{region " SIGNAL AREA : NAME->C_Pnt_Hv_Off LENGTH->2 STARTBIT :22"}
_FB_CanTx_Message_Unpack_450.S_Bit_22		:= (GVL.IOVD.C_Pnt_Hv_Off.x OR GVL.IOVD.C_Pnt_Hv_Off.na) AND NOT GVL.IOVD.C_Pnt_Hv_Off.e; 
_FB_CanTx_Message_Unpack_450.S_Bit_23		:= NOT GVL.IOVD.C_Pnt_Hv_Off.v OR GVL.IOVD.C_Pnt_Hv_Off.na OR GVL.IOVD.C_Pnt_Hv_Off.e; 
{endregion}

{region " SIGNAL AREA : NAME->C_Bat_Lo_Hv_Off LENGTH->2 STARTBIT :24"}
_FB_CanTx_Message_Unpack_450.S_Bit_24		:= (GVL.IOVD.C_Bat_Lo_Hv_Off.x OR GVL.IOVD.C_Bat_Lo_Hv_Off.na) AND NOT GVL.IOVD.C_Bat_Lo_Hv_Off.e; 
_FB_CanTx_Message_Unpack_450.S_Bit_25		:= NOT GVL.IOVD.C_Bat_Lo_Hv_Off.v OR GVL.IOVD.C_Bat_Lo_Hv_Off.na OR GVL.IOVD.C_Bat_Lo_Hv_Off.e; 
{endregion}

{region " SIGNAL AREA : NAME->C_Tm_Hv_Off LENGTH->2 STARTBIT :26"}
_FB_CanTx_Message_Unpack_450.S_Bit_26		:= (GVL.IOVD.C_Tm_Hv_Off.x OR GVL.IOVD.C_Tm_Hv_Off.na) AND NOT GVL.IOVD.C_Tm_Hv_Off.e; 
_FB_CanTx_Message_Unpack_450.S_Bit_27		:= NOT GVL.IOVD.C_Tm_Hv_Off.v OR GVL.IOVD.C_Tm_Hv_Off.na OR GVL.IOVD.C_Tm_Hv_Off.e; 
{endregion}

{region " SIGNAL AREA : NAME->C_Diag_Hv_Off LENGTH->2 STARTBIT :28"}
_FB_CanTx_Message_Unpack_450.S_Bit_28		:= (GVL.IOVD.C_Diag_Hv_Off.x OR GVL.IOVD.C_Diag_Hv_Off.na) AND NOT GVL.IOVD.C_Diag_Hv_Off.e; 
_FB_CanTx_Message_Unpack_450.S_Bit_29		:= NOT GVL.IOVD.C_Diag_Hv_Off.v OR GVL.IOVD.C_Diag_Hv_Off.na OR GVL.IOVD.C_Diag_Hv_Off.e; 
{endregion}

{region " SIGNAL AREA : NAME->C_Hv_On LENGTH->2 STARTBIT :32"}
_FB_CanTx_Message_Unpack_450.S_Bit_32		:= (GVL.IOVD.C_Hv_On.x OR GVL.IOVD.C_Hv_On.na) AND NOT GVL.IOVD.C_Hv_On.e; 
_FB_CanTx_Message_Unpack_450.S_Bit_33		:= NOT GVL.IOVD.C_Hv_On.v OR GVL.IOVD.C_Hv_On.na OR GVL.IOVD.C_Hv_On.e; 
{endregion}

{region " SIGNAL AREA : NAME->C_Hv_Off LENGTH->2 STARTBIT :34"}
_FB_CanTx_Message_Unpack_450.S_Bit_34		:= (GVL.IOVD.C_Hv_Off.x OR GVL.IOVD.C_Hv_Off.na) AND NOT GVL.IOVD.C_Hv_Off.e; 
_FB_CanTx_Message_Unpack_450.S_Bit_35		:= NOT GVL.IOVD.C_Hv_Off.v OR GVL.IOVD.C_Hv_Off.na OR GVL.IOVD.C_Hv_Off.e; 
{endregion}

{region " SIGNAL AREA : NAME->S_Hv_On_Prc LENGTH->2 STARTBIT :36"}
_FB_CanTx_Message_Unpack_450.S_Bit_36		:= (GVL.IOVD.S_Hv_On_Prc.x OR GVL.IOVD.S_Hv_On_Prc.na) AND NOT GVL.IOVD.S_Hv_On_Prc.e; 
_FB_CanTx_Message_Unpack_450.S_Bit_37		:= NOT GVL.IOVD.S_Hv_On_Prc.v OR GVL.IOVD.S_Hv_On_Prc.na OR GVL.IOVD.S_Hv_On_Prc.e; 
{endregion}

{region " SIGNAL AREA : NAME->S_Hv_Off_Prc LENGTH->2 STARTBIT :38"}
_FB_CanTx_Message_Unpack_450.S_Bit_38		:= (GVL.IOVD.S_Hv_Off_Prc.x OR GVL.IOVD.S_Hv_Off_Prc.na) AND NOT GVL.IOVD.S_Hv_Off_Prc.e; 
_FB_CanTx_Message_Unpack_450.S_Bit_39		:= NOT GVL.IOVD.S_Hv_Off_Prc.v OR GVL.IOVD.S_Hv_Off_Prc.na OR GVL.IOVD.S_Hv_Off_Prc.e; 
{endregion}

{region " SIGNAL AREA : NAME->S_Em_Stop LENGTH->2 STARTBIT :40"}
_FB_CanTx_Message_Unpack_450.S_Bit_40		:= (GVL.IOVD.S_Em_Stop.x OR GVL.IOVD.S_Em_Stop.na) AND NOT GVL.IOVD.S_Em_Stop.e; 
_FB_CanTx_Message_Unpack_450.S_Bit_41		:= NOT GVL.IOVD.S_Em_Stop.v OR GVL.IOVD.S_Em_Stop.na OR GVL.IOVD.S_Em_Stop.e; 
{endregion}

{region " SIGNAL AREA : NAME->S_Hv_On_En LENGTH->2 STARTBIT :42"}
_FB_CanTx_Message_Unpack_450.S_Bit_42		:= (GVL.IOVD.S_Hv_On_En.x OR GVL.IOVD.S_Hv_On_En.na) AND NOT GVL.IOVD.S_Hv_On_En.e; 
_FB_CanTx_Message_Unpack_450.S_Bit_43		:= NOT GVL.IOVD.S_Hv_On_En.v OR GVL.IOVD.S_Hv_On_En.na OR GVL.IOVD.S_Hv_On_En.e; 
{endregion}

{region " SIGNAL AREA : NAME->S_Hv_Off_En LENGTH->2 STARTBIT :44"}
_FB_CanTx_Message_Unpack_450.S_Bit_44		:= (GVL.IOVD.S_Hv_Off_En.x OR GVL.IOVD.S_Hv_Off_En.na) AND NOT GVL.IOVD.S_Hv_Off_En.e; 
_FB_CanTx_Message_Unpack_450.S_Bit_45		:= NOT GVL.IOVD.S_Hv_Off_En.v OR GVL.IOVD.S_Hv_Off_En.na OR GVL.IOVD.S_Hv_Off_En.e; 
{endregion}

{region " SIGNAL AREA : NAME->C_Mn_Ct_On LENGTH->2 STARTBIT :46"}
_FB_CanTx_Message_Unpack_450.S_Bit_46		:= (GVL.IOVD.C_Mn_Ct_On.x OR GVL.IOVD.C_Mn_Ct_On.na) AND NOT GVL.IOVD.C_Mn_Ct_On.e; 
_FB_CanTx_Message_Unpack_450.S_Bit_47		:= NOT GVL.IOVD.C_Mn_Ct_On.v OR GVL.IOVD.C_Mn_Ct_On.na OR GVL.IOVD.C_Mn_Ct_On.e; 
{endregion}

{region " SIGNAL AREA : NAME->S_Mn_Ct LENGTH->2 STARTBIT :48"}
_FB_CanTx_Message_Unpack_450.S_Bit_48		:= (GVL.IOVD.S_Mn_Ct.x OR GVL.IOVD.S_Mn_Ct.na) AND NOT GVL.IOVD.S_Mn_Ct.e; 
_FB_CanTx_Message_Unpack_450.S_Bit_49		:= NOT GVL.IOVD.S_Mn_Ct.v OR GVL.IOVD.S_Mn_Ct.na OR GVL.IOVD.S_Mn_Ct.e; 
{endregion}

{region " SIGNAL AREA : NAME->C_Prechrg_Ct_On LENGTH->2 STARTBIT :50"}
_FB_CanTx_Message_Unpack_450.S_Bit_50		:= (GVL.IOVD.C_Prechrg_Ct_On.x OR GVL.IOVD.C_Prechrg_Ct_On.na) AND NOT GVL.IOVD.C_Prechrg_Ct_On.e; 
_FB_CanTx_Message_Unpack_450.S_Bit_51		:= NOT GVL.IOVD.C_Prechrg_Ct_On.v OR GVL.IOVD.C_Prechrg_Ct_On.na OR GVL.IOVD.C_Prechrg_Ct_On.e; 
{endregion}

{region " SIGNAL AREA : NAME->S_Prechrg_Ct LENGTH->2 STARTBIT :52"}
_FB_CanTx_Message_Unpack_450.S_Bit_52		:= (GVL.IOVD.S_Prechrg_Ct.x OR GVL.IOVD.S_Prechrg_Ct.na) AND NOT GVL.IOVD.S_Prechrg_Ct.e; 
_FB_CanTx_Message_Unpack_450.S_Bit_53		:= NOT GVL.IOVD.S_Prechrg_Ct.v OR GVL.IOVD.S_Prechrg_Ct.na OR GVL.IOVD.S_Prechrg_Ct.e; 
{endregion}

{region " SIGNAL AREA : NAME->S_ER_HV LENGTH->2 STARTBIT :54"}
_FB_CanTx_Message_Unpack_450.S_Bit_54		:= (GVL.IOVD.S_ER_HV.x OR GVL.IOVD.S_ER_HV.na) AND NOT GVL.IOVD.S_ER_HV.e; 
_FB_CanTx_Message_Unpack_450.S_Bit_55		:= NOT GVL.IOVD.S_ER_HV.v OR GVL.IOVD.S_ER_HV.na OR GVL.IOVD.S_ER_HV.e; 
{endregion}

{region " SIGNAL AREA : NAME->S_ER_Mn_Ct LENGTH->2 STARTBIT :56"}
_FB_CanTx_Message_Unpack_450.S_Bit_56		:= (GVL.IOVD.S_ER_Mn_Ct.x OR GVL.IOVD.S_ER_Mn_Ct.na) AND NOT GVL.IOVD.S_ER_Mn_Ct.e; 
_FB_CanTx_Message_Unpack_450.S_Bit_57		:= NOT GVL.IOVD.S_ER_Mn_Ct.v OR GVL.IOVD.S_ER_Mn_Ct.na OR GVL.IOVD.S_ER_Mn_Ct.e; 

{endregion}

{region " SIGNAL AREA : NAME->S_ER_Prechrg_Ct LENGTH->2 STARTBIT :58"}
_FB_CanTx_Message_Unpack_450.S_Bit_58		:= (GVL.IOVD.S_ER_Prechrg_Ct.x OR GVL.IOVD.S_ER_Prechrg_Ct.na) AND NOT GVL.IOVD.S_ER_Prechrg_Ct.e; 
_FB_CanTx_Message_Unpack_450.S_Bit_59		:= NOT GVL.IOVD.S_ER_Prechrg_Ct.v OR GVL.IOVD.S_ER_Prechrg_Ct.na OR GVL.IOVD.S_ER_Prechrg_Ct.e; 
{endregion}

{region " SIGNAL AREA : NAME->S_Hv_On LENGTH->2 STARTBIT :60"}
_FB_CanTx_Message_Unpack_450.S_Bit_60		:= (GVL.IOVD.S_Hv_On.x OR GVL.IOVD.S_Hv_On.na) AND NOT GVL.IOVD.S_Hv_On.e; 
_FB_CanTx_Message_Unpack_450.S_Bit_61		:= NOT GVL.IOVD.S_Hv_On.v OR GVL.IOVD.S_Hv_On.na OR GVL.IOVD.S_Hv_On.e; 
{endregion}

{region " SIGNAL AREA : NAME->S_HV_HVAC_En LENGTH->2 STARTBIT :62"}
_FB_CanTx_Message_Unpack_450.S_Bit_62		:= (GVL.IOVD.S_HV_HVAC_En.x OR GVL.IOVD.S_HV_HVAC_En.na) AND NOT GVL.IOVD.S_HV_HVAC_En.e;
_FB_CanTx_Message_Unpack_450.S_Bit_63		:= NOT GVL.IOVD.S_HV_HVAC_En.v OR GVL.IOVD.S_HV_HVAC_En.na OR GVL.IOVD.S_HV_HVAC_En.e;
{endregion}

_FB_CanTx_Message_Unpack_450.S_Bit_2	:= TRUE;
_FB_CanTx_Message_Unpack_450.S_Bit_3	:= TRUE;
_FB_CanTx_Message_Unpack_450.S_Bit_4	:= TRUE;
_FB_CanTx_Message_Unpack_450.S_Bit_5	:= TRUE;
_FB_CanTx_Message_Unpack_450.S_Bit_14	:= TRUE;
_FB_CanTx_Message_Unpack_450.S_Bit_15	:= TRUE;
_FB_CanTx_Message_Unpack_450.S_Bit_18	:= TRUE;
_FB_CanTx_Message_Unpack_450.S_Bit_19	:= TRUE;
_FB_CanTx_Message_Unpack_450.S_Bit_20	:= TRUE;
_FB_CanTx_Message_Unpack_450.S_Bit_21	:= TRUE;
_FB_CanTx_Message_Unpack_450.S_Bit_30	:= TRUE;
_FB_CanTx_Message_Unpack_450.S_Bit_31	:= TRUE;

_FB_CanTx_Message_Unpack_450 (		C_Enable		:= GVL.IOVD.C_En_HV_Durum_0X450,
     								Obj_CAN			:= ADR(GVL.IC.Obj_CAN0),
     								X_MsgID			:= 16#450,
     								Tm_CycleTime	:= TIME#250MS,
     								N_Msg_Dlc		:= 8,
     								S_Extended		:= 0,
     								S_Sent_Ok   	=> GVL.IOVD.S_SentOk_HV_Durum_0X450);
{endregion}
//-----------------------------------------------------------------------------------------------------------------------------
//-----------------------------------------------------------------------------------------------------------------------------
{region " MESSAGE AREA :TCU_Trolley_Durum- ID:460"}

{region " SIGNAL AREA : NAME->S_Mn_Ct_Req LENGTH->2 STARTBIT :0"}
_FB_CanTx_Message_Unpack_460.S_Bit_0		:= (GVL.IOVD.S_Mn_Ct_Req.x OR GVL.IOVD.S_Mn_Ct_Req.na) AND NOT GVL.IOVD.S_Mn_Ct_Req.e; 
_FB_CanTx_Message_Unpack_460.S_Bit_1		:= NOT GVL.IOVD.S_Mn_Ct_Req.v OR GVL.IOVD.S_Mn_Ct_Req.na OR GVL.IOVD.S_Mn_Ct_Req.e; 
{endregion}

{region " SIGNAL AREA : NAME->S_Sys_On LENGTH->2 STARTBIT :2"}
_FB_CanTx_Message_Unpack_460.S_Bit_2		:= (GVL.IOVD.S_Sys_On.x OR GVL.IOVD.S_Sys_On.na) AND NOT GVL.IOVD.S_Sys_On.e; 
_FB_CanTx_Message_Unpack_460.S_Bit_3		:= NOT GVL.IOVD.S_Sys_On.v OR GVL.IOVD.S_Sys_On.na OR GVL.IOVD.S_Sys_On.e; 
{endregion}

{region " SIGNAL AREA : NAME->S_Mot_Cnv_On_Req LENGTH->2 STARTBIT :4"}
_FB_CanTx_Message_Unpack_460.S_Bit_4		:= (GVL.IOVD.S_Mot_Cnv_On_Req.x OR GVL.IOVD.S_Mot_Cnv_On_Req.na) AND NOT GVL.IOVD.S_Mot_Cnv_On_Req.e; 
_FB_CanTx_Message_Unpack_460.S_Bit_5		:= NOT GVL.IOVD.S_Mot_Cnv_On_Req.v OR GVL.IOVD.S_Mot_Cnv_On_Req.na OR GVL.IOVD.S_Mot_Cnv_On_Req.e; 

{endregion}

{region " SIGNAL AREA : NAME->S_Mot_Cnv_On LENGTH->2 STARTBIT :6"}
_FB_CanTx_Message_Unpack_460.S_Bit_6		:= (GVL.IOVD.S_Mot_Cnv_On.x OR GVL.IOVD.S_Mot_Cnv_On.na) AND NOT GVL.IOVD.S_Mot_Cnv_On.e; 
_FB_CanTx_Message_Unpack_460.S_Bit_7		:= NOT GVL.IOVD.S_Mot_Cnv_On.v OR GVL.IOVD.S_Mot_Cnv_On.na OR GVL.IOVD.S_Mot_Cnv_On.e; 

{endregion}

{region " SIGNAL AREA : NAME->S_24V_Bat_Cnv_On_Req LENGTH->2 STARTBIT :8"}
_FB_CanTx_Message_Unpack_460.S_Bit_8		:= (GVL.IOVD.S_24V_Bat_Cnv_On_Req.x OR GVL.IOVD.S_24V_Bat_Cnv_On_Req.na) AND NOT GVL.IOVD.S_24V_Bat_Cnv_On_Req.e; 
_FB_CanTx_Message_Unpack_460.S_Bit_9		:= NOT GVL.IOVD.S_24V_Bat_Cnv_On_Req.v OR GVL.IOVD.S_24V_Bat_Cnv_On_Req.na OR GVL.IOVD.S_24V_Bat_Cnv_On_Req.e; 

{endregion}

{region " SIGNAL AREA : NAME->S_24V_Sp_On LENGTH->2 STARTBIT :10"}
_FB_CanTx_Message_Unpack_460.S_Bit_10		:= (GVL.IOVD.S_24V_Sp_On.x OR GVL.IOVD.S_24V_Sp_On.na) AND NOT GVL.IOVD.S_24V_Sp_On.e; 
_FB_CanTx_Message_Unpack_460.S_Bit_11		:= NOT GVL.IOVD.S_24V_Sp_On.v OR GVL.IOVD.S_24V_Sp_On.na OR GVL.IOVD.S_24V_Sp_On.e; 

{endregion}

{region " SIGNAL AREA : NAME->S_Pnt_Chrg_Req LENGTH->2 STARTBIT :12"}
_FB_CanTx_Message_Unpack_460.S_Bit_12		:= (GVL.IOVD.S_Pnt_Chrg_Req.x OR GVL.IOVD.S_Pnt_Chrg_Req.na) AND NOT GVL.IOVD.S_Pnt_Chrg_Req.e; 
_FB_CanTx_Message_Unpack_460.S_Bit_13		:= NOT GVL.IOVD.S_Pnt_Chrg_Req.v OR GVL.IOVD.S_Pnt_Chrg_Req.na OR GVL.IOVD.S_Pnt_Chrg_Req.e; 

{endregion}

{region " SIGNAL AREA : NAME->S_Pnt_Chrg_Fdbk LENGTH->2 STARTBIT :14"}
_FB_CanTx_Message_Unpack_460.S_Bit_14		:= (GVL.IOVD.S_Pnt_Chrg_Fdbk.x OR GVL.IOVD.S_Pnt_Chrg_Fdbk.na) AND NOT GVL.IOVD.S_Pnt_Chrg_Fdbk.e; 
_FB_CanTx_Message_Unpack_460.S_Bit_15		:= NOT GVL.IOVD.S_Pnt_Chrg_Fdbk.v OR GVL.IOVD.S_Pnt_Chrg_Fdbk.na OR GVL.IOVD.S_Pnt_Chrg_Fdbk.e; 
{endregion}

{region " SIGNAL AREA : NAME->Z_Drv_Dir_Req LENGTH->2 STARTBIT :16"}
_FB_UNPACK_BYTE_TO_8BITS_0 (	S_Bit_0		=> _FB_CanTx_Message_Unpack_460.S_Bit_16,
								S_Bit_1		=> _FB_CanTx_Message_Unpack_460.S_Bit_17 ,
								X_BYTE_0	:=
(*SELECT 1 : Is force active?*)					SEL((GVL.IOVD.Z_Drv_Dir_Req.v AND NOT GVL.IOVD.Z_Drv_Dir_Req.RangeExcd),
(*DEFAULT VALUE assignment*)					0,
(*FORCE is active*)								GVL.IOVD.Z_Drv_Dir_Req.x));
{endregion}

{region " SIGNAL AREA : NAME->Z_Drv_Dir LENGTH->2 STARTBIT :18"}
_FB_UNPACK_BYTE_TO_8BITS_1 (	S_Bit_0		=> _FB_CanTx_Message_Unpack_460.S_Bit_18,
								S_Bit_1		=> _FB_CanTx_Message_Unpack_460.S_Bit_19 ,
								X_BYTE_0	:=
(*SELECT 1 : Is force active?*)					SEL((GVL.IOVD.Z_Drv_Dir.v AND NOT GVL.IOVD.Z_Drv_Dir.RangeExcd),
(*DEFAULT VALUE assignment*)					0,
(*FORCE is active*)								GVL.IOVD.Z_Drv_Dir.x));
{endregion}

{region " SIGNAL AREA : NAME->S_Elec_Mode_Req LENGTH->2 STARTBIT :20"}
_FB_CanTx_Message_Unpack_460.S_Bit_20		:= (GVL.IOVD.S_Elec_Mode_Req.x OR GVL.IOVD.S_Elec_Mode_Req.na) AND NOT GVL.IOVD.S_Elec_Mode_Req.e; 
_FB_CanTx_Message_Unpack_460.S_Bit_21		:= NOT GVL.IOVD.S_Elec_Mode_Req.v OR GVL.IOVD.S_Elec_Mode_Req.na OR GVL.IOVD.S_Elec_Mode_Req.e; 
{endregion}

{region " SIGNAL AREA : NAME->S_Elec_Mode_Actv LENGTH->2 STARTBIT :22"}
_FB_CanTx_Message_Unpack_460.S_Bit_22		:= (GVL.IOVD.S_Elec_Mode_Actv.x OR GVL.IOVD.S_Elec_Mode_Actv.na) AND NOT GVL.IOVD.S_Elec_Mode_Actv.e; 
_FB_CanTx_Message_Unpack_460.S_Bit_23		:= NOT GVL.IOVD.S_Elec_Mode_Actv.v OR GVL.IOVD.S_Elec_Mode_Actv.na OR GVL.IOVD.S_Elec_Mode_Actv.e; 
{endregion}
		  
{region " SIGNAL AREA : NAME->S_Bat_Mode_Req LENGTH->2 STARTBIT :24"}
_FB_CanTx_Message_Unpack_460.S_Bit_24		:= (GVL.IOVD.S_Bat_Mode_Req.x OR GVL.IOVD.S_Bat_Mode_Req.na) AND NOT GVL.IOVD.S_Bat_Mode_Req.e; 
_FB_CanTx_Message_Unpack_460.S_Bit_25		:= NOT GVL.IOVD.S_Bat_Mode_Req.v OR GVL.IOVD.S_Bat_Mode_Req.na OR GVL.IOVD.S_Bat_Mode_Req.e; 
{endregion}

{region " SIGNAL AREA : NAME->S_Bat_Mode_Actv LENGTH->2 STARTBIT :26"}
_FB_CanTx_Message_Unpack_460.S_Bit_26		:= (GVL.IOVD.S_Bat_Mode_Actv.x OR GVL.IOVD.S_Bat_Mode_Actv.na) AND NOT GVL.IOVD.S_Bat_Mode_Actv.e; 
_FB_CanTx_Message_Unpack_460.S_Bit_27		:= NOT GVL.IOVD.S_Bat_Mode_Actv.v OR GVL.IOVD.S_Bat_Mode_Actv.na OR GVL.IOVD.S_Bat_Mode_Actv.e; 
{endregion}

{region " SIGNAL AREA : NAME->S_Elec_Ret_En LENGTH->2 STARTBIT :28"}
_FB_CanTx_Message_Unpack_460.S_Bit_28		:= (GVL.IOVD.S_Elec_Ret_En.x OR GVL.IOVD.S_Elec_Ret_En.na) AND NOT GVL.IOVD.S_Elec_Ret_En.e; 
_FB_CanTx_Message_Unpack_460.S_Bit_29		:= NOT GVL.IOVD.S_Elec_Ret_En.v OR GVL.IOVD.S_Elec_Ret_En.na OR GVL.IOVD.S_Elec_Ret_En.e; 
{endregion}

{region " SIGNAL AREA : NAME->S_Elec_Brk_En LENGTH->2 STARTBIT :30"}
_FB_CanTx_Message_Unpack_460.S_Bit_30		:= (GVL.IOVD.S_Elec_Brk_En.x OR GVL.IOVD.S_Elec_Brk_En.na) AND NOT GVL.IOVD.S_Elec_Brk_En.e; 
_FB_CanTx_Message_Unpack_460.S_Bit_31		:= NOT GVL.IOVD.S_Elec_Brk_En.v OR GVL.IOVD.S_Elec_Brk_En.na OR GVL.IOVD.S_Elec_Brk_En.e; 
{endregion}

{region " SIGNAL AREA : NAME->S_Tintl LENGTH->2 STARTBIT :32"}
_FB_CanTx_Message_Unpack_460.S_Bit_32		:= (GVL.IOVD.S_Tintl.x OR GVL.IOVD.S_Tintl.na) AND NOT GVL.IOVD.S_Tintl.e; 
_FB_CanTx_Message_Unpack_460.S_Bit_33		:= NOT GVL.IOVD.S_Tintl.v OR GVL.IOVD.S_Tintl.na OR GVL.IOVD.S_Tintl.e; 
{endregion}

{region " SIGNAL AREA : NAME->S_Em_Deact LENGTH->2 STARTBIT :34"}
_FB_CanTx_Message_Unpack_460.S_Bit_34		:= (GVL.IOVD.S_Em_Deact.x OR GVL.IOVD.S_Em_Deact.na) AND NOT GVL.IOVD.S_Em_Deact.e; 
_FB_CanTx_Message_Unpack_460.S_Bit_35		:= NOT GVL.IOVD.S_Em_Deact.v OR GVL.IOVD.S_Em_Deact.na OR GVL.IOVD.S_Em_Deact.e; 
{endregion}

{region " SIGNAL AREA : NAME->S_Rs_Cosu_Req LENGTH->2 STARTBIT :36"}
_FB_CanTx_Message_Unpack_460.S_Bit_36		:= (GVL.IOVD.S_Rs_Cosu_Req.x OR GVL.IOVD.S_Rs_Cosu_Req.na) AND NOT GVL.IOVD.S_Rs_Cosu_Req.e; 
_FB_CanTx_Message_Unpack_460.S_Bit_37		:= NOT GVL.IOVD.S_Rs_Cosu_Req.v OR GVL.IOVD.S_Rs_Cosu_Req.na OR GVL.IOVD.S_Rs_Cosu_Req.e; 
{endregion}

{region " SIGNAL AREA : NAME->S_TCU_Hlt_Brk_Req LENGTH->2 STARTBIT :38"}
_FB_CanTx_Message_Unpack_460.S_Bit_38		:= (GVL.IOVD.S_TCU_Hlt_Brk_Req.x OR GVL.IOVD.S_TCU_Hlt_Brk_Req.na) AND NOT GVL.IOVD.S_TCU_Hlt_Brk_Req.e; 
_FB_CanTx_Message_Unpack_460.S_Bit_39		:= NOT GVL.IOVD.S_TCU_Hlt_Brk_Req.v OR GVL.IOVD.S_TCU_Hlt_Brk_Req.na OR GVL.IOVD.S_TCU_Hlt_Brk_Req.e; 

{endregion}

{region " SIGNAL AREA : NAME->S_Insu_Test_Mod_Actv LENGTH->2 STARTBIT :40"}
_FB_CanTx_Message_Unpack_460.S_Bit_40		:= (GVL.IOVD.S_Insu_Test_Mod_Actv.x OR GVL.IOVD.S_Insu_Test_Mod_Actv.na) AND NOT GVL.IOVD.S_Insu_Test_Mod_Actv.e; 
_FB_CanTx_Message_Unpack_460.S_Bit_41		:= NOT GVL.IOVD.S_Insu_Test_Mod_Actv.v OR GVL.IOVD.S_Insu_Test_Mod_Actv.na OR GVL.IOVD.S_Insu_Test_Mod_Actv.e; 

{endregion}

{region " SIGNAL AREA : NAME->S_Engy_Flw_Trol LENGTH->2 STARTBIT :42"}
_FB_CanTx_Message_Unpack_460.S_Bit_42		:= (GVL.IOVD.S_Engy_Flw_Trol.x OR GVL.IOVD.S_Engy_Flw_Trol.na) AND NOT GVL.IOVD.S_Engy_Flw_Trol.e; 
_FB_CanTx_Message_Unpack_460.S_Bit_43		:= NOT GVL.IOVD.S_Engy_Flw_Trol.v OR GVL.IOVD.S_Engy_Flw_Trol.na OR GVL.IOVD.S_Engy_Flw_Trol.e; 

{endregion}

{region " SIGNAL AREA : NAME->S_Engy_Flw_Bat LENGTH->2 STARTBIT :44"}
_FB_CanTx_Message_Unpack_460.S_Bit_44		:= (GVL.IOVD.S_Engy_Flw_Bat.x OR GVL.IOVD.S_Engy_Flw_Bat.na) AND NOT GVL.IOVD.S_Engy_Flw_Bat.e; 
_FB_CanTx_Message_Unpack_460.S_Bit_45		:= NOT GVL.IOVD.S_Engy_Flw_Bat.v OR GVL.IOVD.S_Engy_Flw_Bat.na OR GVL.IOVD.S_Engy_Flw_Bat.e; 

{endregion}
		  
{region " SIGNAL AREA : NAME->S_Trol_Volt_Actv LENGTH->2 STARTBIT :46"}
_FB_CanTx_Message_Unpack_460.S_Bit_46		:= (GVL.IOVD.S_Trol_Volt_Actv.x OR GVL.IOVD.S_Trol_Volt_Actv.na) AND NOT GVL.IOVD.S_Trol_Volt_Actv.e; 
_FB_CanTx_Message_Unpack_460.S_Bit_47		:= NOT GVL.IOVD.S_Trol_Volt_Actv.v OR GVL.IOVD.S_Trol_Volt_Actv.na OR GVL.IOVD.S_Trol_Volt_Actv.e; 

{endregion}			   
		  
{region " SIGNAL AREA : NAME->C_Mot_Fan_Ct LENGTH->2 STARTBIT :48"}
_FB_CanTx_Message_Unpack_460.S_Bit_48		:= (GVL.IOVD.C_Mot_Fan_Ct.x OR GVL.IOVD.C_Mot_Fan_Ct.na) AND NOT GVL.IOVD.C_Mot_Fan_Ct.e; 
_FB_CanTx_Message_Unpack_460.S_Bit_49		:= NOT GVL.IOVD.C_Mot_Fan_Ct.v OR GVL.IOVD.C_Mot_Fan_Ct.na OR GVL.IOVD.C_Mot_Fan_Ct.e; 

{endregion}	
		  
{region " SIGNAL AREA : NAME->S_Mot_Fan_Thrm_Ct LENGTH->2 STARTBIT :50"}
_FB_CanTx_Message_Unpack_460.S_Bit_50		:= (GVL.IOVD.S_Mot_Fan_Thrm_Ct.x OR GVL.IOVD.S_Mot_Fan_Thrm_Ct.na) AND NOT GVL.IOVD.S_Mot_Fan_Thrm_Ct.e; 
_FB_CanTx_Message_Unpack_460.S_Bit_51		:= NOT GVL.IOVD.S_Mot_Fan_Thrm_Ct.v OR GVL.IOVD.S_Mot_Fan_Thrm_Ct.na OR GVL.IOVD.S_Mot_Fan_Thrm_Ct.e; 

{endregion}		

{region " SIGNAL AREA : NAME->S_ER_Elec_Brk_Amb LENGTH->2 STARTBIT :52"}
_FB_CanTx_Message_Unpack_460.S_Bit_52		:= (GVL.IOVD.S_ER_Elec_Brk_Amb.x OR GVL.IOVD.S_ER_Elec_Brk_Amb.na) AND NOT GVL.IOVD.S_ER_Elec_Brk_Amb.e; 
_FB_CanTx_Message_Unpack_460.S_Bit_53		:= NOT GVL.IOVD.S_ER_Elec_Brk_Amb.v OR GVL.IOVD.S_ER_Elec_Brk_Amb.na OR GVL.IOVD.S_ER_Elec_Brk_Amb.e; 

{endregion}

{region " SIGNAL AREA : NAME->S_ER_Elec_Brk_Red LENGTH->2 STARTBIT :54"}
_FB_CanTx_Message_Unpack_460.S_Bit_54		:= (GVL.IOVD.S_ER_Elec_Brk_Red.x OR GVL.IOVD.S_ER_Elec_Brk_Red.na) AND NOT GVL.IOVD.S_ER_Elec_Brk_Red.e; 
_FB_CanTx_Message_Unpack_460.S_Bit_55		:= NOT GVL.IOVD.S_ER_Elec_Brk_Red.v OR GVL.IOVD.S_ER_Elec_Brk_Red.na OR GVL.IOVD.S_ER_Elec_Brk_Red.e; 
{endregion}	  
 
_FB_CanTx_Message_Unpack_460.X_Byte_7		:=	SEL((GVL.IOVD.Z_Mc_Stat.v AND NOT GVL.IOVD.Z_Mc_Stat.RangeExcd),
(*SELECT 2 : Is NOT AVAILABLE ?*)				SEL(GVL.IOVD.Z_Mc_Stat.na,
(*SELECT 3 : Is ERROR active ?*)				SEL(GVL.IOVD.Z_Mc_Stat.e,
(*DEFAULT VALUE assignment*)					0,
(*ERROR is active*)								16#FE),
(*NOT AVAILABLE is active*)						16#FF),
(*Transmission is VALID*)						USINT_TO_BYTE(REAL_TO_USINT((GVL.IOVD.Z_Mc_Stat.x))));
	 
_FB_CanTx_Message_Unpack_460 (	C_Enable		:= GVL.IOVD.C_En_TCU_Trolleybus_Durum_0X460,
     							Obj_CAN			:= ADR(GVL.IC.Obj_CAN0),
     							X_MsgID			:= 16#460,
     							Tm_CycleTime	:= TIME#250MS,
     							N_Msg_Dlc		:= 8,
     							S_Extended		:= 0,
     							S_Sent_Ok   	=> GVL.IOVD.S_SentOk_TCU_Trolleybus_Durum_0X460);
{endregion}
//-----------------------------------------------------------------------------------------------------------------------------
//-----------------------------------------------------------------------------------------------------------------------------
{region " MESSAGE AREA :TCU_Surus_Limit- ID:462"}

{region " SIGNAL AREA : NAME->X_Spd_Max_Fwd LENGTH->8 STARTBIT :0"}
_FB_CanTx_Message_Unpack_462.X_Byte_0		:=
(*SELECT 1 : Is data valid and range is not exceed?*)	SEL((GVL.IOVD.X_Spd_Max_Fwd.v AND NOT GVL.IOVD.X_Spd_Max_Fwd.RangeExcd),
(*SELECT 2 : Is NOT AVAILABLE ?*)						SEL(GVL.IOVD.X_Spd_Max_Fwd.na,
(*SELECT 3 : Is ERROR active ?*)						SEL(GVL.IOVD.X_Spd_Max_Fwd.e,
(*DEFAULT VALUE assignment*)							0,
(*ERROR is active*)										16#FE),
(*NOT AVAILABLE is active*)								16#FF),
(*Transmission is VALID*)								USINT_TO_BYTE(REAL_TO_USINT((GVL.IOVD.X_Spd_Max_Fwd.x))));
{endregion}

{region " SIGNAL AREA : NAME->X_Spd_Max_Bwd LENGTH->8 STARTBIT :8"}
_FB_CanTx_Message_Unpack_462.X_Byte_1		:=
(*SELECT 1 : Is data valid and range is not exceed?*)	SEL((GVL.IOVD.X_Spd_Max_Bwd.v AND NOT GVL.IOVD.X_Spd_Max_Bwd.RangeExcd),
(*SELECT 2 : Is NOT AVAILABLE ?*)						SEL(GVL.IOVD.X_Spd_Max_Bwd.na,
(*SELECT 3 : Is ERROR active ?*)						SEL(GVL.IOVD.X_Spd_Max_Bwd.e,
(*DEFAULT VALUE assignment*)							0,
(*ERROR is active*)										16#FE),
(*NOT AVAILABLE is active*)								16#FF),
(*Transmission is VALID*)								USINT_TO_BYTE(REAL_TO_USINT((GVL.IOVD.X_Spd_Max_Bwd.x))));
{endregion}

{region " SIGNAL AREA : NAME->X_Ang_Str LENGTH->8 STARTBIT :16"}
_FB_CanTx_Message_Unpack_462.X_Byte_2		:=
(*SELECT 1 : Is data valid and range is not exceed?*)	SEL((GVL.IOVD.X_Ang_Str.v AND NOT GVL.IOVD.X_Ang_Str.RangeExcd),
(*SELECT 2 : Is NOT AVAILABLE ?*)						SEL(GVL.IOVD.X_Ang_Str.na,
(*SELECT 3 : Is ERROR active ?*)						SEL(GVL.IOVD.X_Ang_Str.e,
(*DEFAULT VALUE assignment*)							USINT_TO_BYTE(REAL_TO_USINT((125))),
(*ERROR is active*)										16#FE),
(*NOT AVAILABLE is active*)								16#FF),
(*Transmission is VALID*)								USINT_TO_BYTE(REAL_TO_USINT((GVL.IOVD.X_Ang_Str.x + 125))));
{endregion}

{region " SIGNAL AREA : NAME->X_Pct_Brk_Pdl LENGTH->8 STARTBIT :32"}
_FB_CanTx_Message_Unpack_462.X_Byte_4		:=
(*SELECT 1 : Is data valid and range is not exceed?*)	SEL((GVL.IOVD.X_Pct_Brk_Pdl.v AND NOT GVL.IOVD.X_Pct_Brk_Pdl.RangeExcd),
(*SELECT 2 : Is NOT AVAILABLE ?*)						SEL(GVL.IOVD.X_Pct_Brk_Pdl.na,
(*SELECT 3 : Is ERROR active ?*)						SEL(GVL.IOVD.X_Pct_Brk_Pdl.e,
(*DEFAULT VALUE assignment*)							0,
(*ERROR is active*)										16#FE),
(*NOT AVAILABLE is active*)								16#FF),
(*Transmission is VALID*)								USINT_TO_BYTE(REAL_TO_USINT((GVL.IOVD.X_Pct_Brk_Pdl.x)/0.4)));
{endregion}

{region " SIGNAL AREA : NAME->X_Pct_Acc_Pdl LENGTH->8 STARTBIT :40"}
_FB_CanTx_Message_Unpack_462.X_Byte_5		:=
(*SELECT 1 : Is data valid and range is not exceed?*)	SEL((GVL.IOVD.X_Pct_Acc_Pdl.v AND NOT GVL.IOVD.X_Pct_Acc_Pdl.RangeExcd),
(*SELECT 2 : Is NOT AVAILABLE ?*)						SEL(GVL.IOVD.X_Pct_Acc_Pdl.na,
(*SELECT 3 : Is ERROR active ?*)						SEL(GVL.IOVD.X_Pct_Acc_Pdl.e,
(*DEFAULT VALUE assignment*)							 0 ,
(*ERROR is active*)										16#FE),
(*NOT AVAILABLE is active*)								16#FF),
(*Transmission is VALID*)								USINT_TO_BYTE(REAL_TO_USINT((GVL.IOVD.X_Pct_Acc_Pdl.x)/0.4)));
{endregion}

{region " SIGNAL AREA : NAME->S_Hlt_Brk_Actv LENGTH->2 STARTBIT :48"}
_FB_CanTx_Message_Unpack_462.S_Bit_48		:=	 (GVL.IOVD.S_Hlt_Brk_Actv.x OR GVL.IOVD.S_Hlt_Brk_Actv.na) AND NOT GVL.IOVD.S_Hlt_Brk_Actv.e; 
_FB_CanTx_Message_Unpack_462.S_Bit_49		:=	 NOT GVL.IOVD.S_Hlt_Brk_Actv.v OR GVL.IOVD.S_Hlt_Brk_Actv.na OR GVL.IOVD.S_Hlt_Brk_Actv.e; 
{endregion}

_FB_CanTx_Message_Unpack_462.X_Byte_3		:= 16#FF;
_FB_CanTx_Message_Unpack_462.S_Bit_50		:= FALSE;
_FB_CanTx_Message_Unpack_462.S_Bit_51		:= FALSE;
_FB_CanTx_Message_Unpack_462.S_Bit_52		:= FALSE;
_FB_CanTx_Message_Unpack_462.S_Bit_53		:= FALSE;
_FB_CanTx_Message_Unpack_462.S_Bit_54		:= FALSE;
_FB_CanTx_Message_Unpack_462.S_Bit_55		:= FALSE;
_FB_CanTx_Message_Unpack_462.X_Byte_7		:= 16#FF;
	 
_FB_CanTx_Message_Unpack_462 (	C_Enable		:= GVL.IOVD.C_En_TCU_Surus_Limit_0X462,
     							Obj_CAN			:= ADR(GVL.IC.Obj_CAN0),
     							X_MsgID			:= 16#462,
     							Tm_CycleTime	:= TIME#250MS,
     							N_Msg_Dlc		:= 8,
     							S_Extended		:= 0,
     							S_Sent_Ok   	=> GVL.IOVD.S_SentOk_TCU_Surus_Limit_0X462);
{endregion}
//-----------------------------------------------------------------------------------------------------------------------------
//-----------------------------------------------------------------------------------------------------------------------------
{region " MESSAGE AREA :TCU_Analog- ID:463"}

{region " SIGNAL AREA : NAME->X_T_Mot LENGTH->8 STARTBIT :0"}
_FB_CanTx_Message_463.X_Byte_0		:=
(*SELECT 1 : Is data valid and range is not exceed?*)	SEL((GVL.IOVD.X_T_Mot.v AND NOT GVL.IOVD.X_T_Mot.RangeExcd),
(*SELECT 2 : Is NOT AVAILABLE ?*)						SEL(GVL.IOVD.X_T_Mot.na,
(*SELECT 3 : Is ERROR active ?*)						SEL(GVL.IOVD.X_T_Mot.e,
(*DEFAULT VALUE assignment*)							USINT_TO_BYTE(REAL_TO_USINT((40))),
(*ERROR is active*)										16#FE),
(*NOT AVAILABLE is active*)								16#FF),
(*Transmission is VALID*)								USINT_TO_BYTE(REAL_TO_USINT((GVL.IOVD.X_T_Mot.x + 40))));
{endregion}

{region " SIGNAL AREA : NAME->X_T_Mot_Cnv LENGTH->8 STARTBIT :8"}
_FB_CanTx_Message_463.X_Byte_1		:=
(*SELECT 1 : Is data valid and range is not exceed?*)	SEL((GVL.IOVD.X_T_Mot_Cnv.v AND NOT GVL.IOVD.X_T_Mot_Cnv.RangeExcd),
(*SELECT 2 : Is NOT AVAILABLE ?*)						SEL(GVL.IOVD.X_T_Mot_Cnv.na,
(*SELECT 3 : Is ERROR active ?*)						SEL(GVL.IOVD.X_T_Mot_Cnv.e,
(*DEFAULT VALUE assignment*)							USINT_TO_BYTE(REAL_TO_USINT((40))),
(*ERROR is active*)										16#FE),
(*NOT AVAILABLE is active*)								16#FF),
(*Transmission is VALID*)								USINT_TO_BYTE(REAL_TO_USINT((GVL.IOVD.X_T_Mot_Cnv.x + 40))));
{endregion}

{region " SIGNAL AREA : NAME->X_T_TCU_Box LENGTH->8 STARTBIT :16"}
_FB_CanTx_Message_463.X_Byte_2		:=
(*SELECT 1 : Is data valid and range is not exceed?*)	SEL((GVL.IOVD.X_T_TCU_Box.v AND NOT GVL.IOVD.X_T_TCU_Box.RangeExcd),
(*SELECT 2 : Is NOT AVAILABLE ?*)						SEL(GVL.IOVD.X_T_TCU_Box.na,
(*SELECT 3 : Is ERROR active ?*)						SEL(GVL.IOVD.X_T_TCU_Box.e,
(*DEFAULT VALUE assignment*)							USINT_TO_BYTE(REAL_TO_USINT((40))),
(*ERROR is active*)										16#FE),
(*NOT AVAILABLE is active*)								16#FF),
(*Transmission is VALID*)								USINT_TO_BYTE(REAL_TO_USINT((GVL.IOVD.X_T_TCU_Box.x + 40))));
{endregion}

{region " SIGNAL AREA : NAME->X_P_ESS LENGTH->16 STARTBIT :32"}
_FB_UNPACK_WORD_TO_BYTE_5 (
		X_WORD_0										:= 
(*SELECT 1 : Is data valid and range is not exceed?*)	SEL((GVL.IOVD.X_P_ESS.v AND NOT GVL.IOVD.X_P_ESS.RangeExcd),
(*SELECT 2 : Is NOT AVAILABLE ?*)						SEL(GVL.IOVD.X_P_ESS.na,
(*SELECT 3 : Is ERROR active ?*)						SEL(GVL.IOVD.X_P_ESS.e,
(*DEFAULT VALUE assignment*)							UINT_TO_WORD(REAL_TO_UINT((3276.6)/0.1)),
(*ERROR is active*)										16#FEFE),
(*NOT AVAILABLE is active*)								16#FFFF),
(*Transmission is VALID*)								UINT_TO_WORD(REAL_TO_UINT((GVL.IOVD.X_P_ESS.x + 3276.6)/0.1))),
		X_BYTE_0										=> _FB_CanTx_Message_463.X_Byte_4,
		X_BYTE_1										=> _FB_CanTx_Message_463.X_Byte_5);
{endregion}

{region " SIGNAL AREA : NAME->X_I_Out_ESS LENGTH->16 STARTBIT :48"}
_FB_UNPACK_WORD_TO_BYTE_6 (
		X_WORD_0										:= 
(*SELECT 1 : Is data valid and range is not exceed?*)	SEL((GVL.IOVD.X_I_Out_ESS.v AND NOT GVL.IOVD.X_I_Out_ESS.RangeExcd),
(*SELECT 2 : Is NOT AVAILABLE ?*)						SEL(GVL.IOVD.X_I_Out_ESS.na,
(*SELECT 3 : Is ERROR active ?*)						SEL(GVL.IOVD.X_I_Out_ESS.e,
(*DEFAULT VALUE assignment*)							UINT_TO_WORD(REAL_TO_UINT((32766))),
(*ERROR is active*)										16#FEFE),
(*NOT AVAILABLE is active*)								16#FFFF),
(*Transmission is VALID*)								UINT_TO_WORD(REAL_TO_UINT((GVL.IOVD.X_I_Out_ESS.x + 32766)))),
		X_BYTE_0										=> _FB_CanTx_Message_463.X_Byte_6,
		X_BYTE_1										=> _FB_CanTx_Message_463.X_Byte_7);
{endregion}

_FB_CanTx_Message_463.X_Byte_3 		:= 16#FF;

_FB_CanTx_Message_463 (		C_Enable		:= GVL.IOVD.C_En_TCU_Analog_0X463,
     						Obj_CAN			:= ADR(GVL.IC.Obj_CAN0),
     						X_MsgID			:= 16#463,
     						Tm_CycleTime	:= TIME#250MS,
     						N_Msg_Dlc		:= 8,
     						S_Extended		:= 0,
     						S_Sent_Ok   	=> GVL.IOVD.S_SentOk_TCU_Analog_0X463);
{endregion}
//-----------------------------------------------------------------------------------------------------------------------------
//-----------------------------------------------------------------------------------------------------------------------------
{region " MESSAGE AREA :TCU_Cikis_Akim_Guc- ID:464"}

{region " SIGNAL AREA : NAME->X_I_Out_Mot_Cnv LENGTH->16 STARTBIT :0"}
_FB_UNPACK_WORD_TO_BYTE_7(
		X_WORD_0										:= 
(*SELECT 1 : Is data valid and range is not exceed?*)	SEL((GVL.IOVD.X_I_Out_Mot_Cnv.v AND NOT GVL.IOVD.X_I_Out_Mot_Cnv.RangeExcd),
(*SELECT 2 : Is NOT AVAILABLE ?*)						SEL(GVL.IOVD.X_I_Out_Mot_Cnv.na,
(*SELECT 3 : Is ERROR active ?*)						SEL(GVL.IOVD.X_I_Out_Mot_Cnv.e,
(*DEFAULT VALUE assignment*)							UINT_TO_WORD(REAL_TO_UINT((1600)/0.05)),
(*ERROR is active*)										16#FEFE),
(*NOT AVAILABLE is active*)								16#FFFF),
(*Transmission is VALID*)								UINT_TO_WORD(REAL_TO_UINT((GVL.IOVD.X_I_Out_Mot_Cnv.x + 1600)/0.05))),
		X_BYTE_0										=> _FB_CanTx_Message_464.X_Byte_0,
		X_BYTE_1										=> _FB_CanTx_Message_464.X_Byte_1);
{endregion}

{region " SIGNAL AREA : NAME->X_I_Brk_Rsr LENGTH->16 STARTBIT :16"}
_FB_UNPACK_WORD_TO_BYTE_8(
		X_WORD_0										:= 
(*SELECT 1 : Is data valid and range is not exceed?*)	SEL((GVL.IOVD.X_I_Brk_Rsr.v AND NOT GVL.IOVD.X_I_Brk_Rsr.RangeExcd),
(*SELECT 2 : Is NOT AVAILABLE ?*)						SEL(GVL.IOVD.X_I_Brk_Rsr.na,
(*SELECT 3 : Is ERROR active ?*)						SEL(GVL.IOVD.X_I_Brk_Rsr.e,
(*DEFAULT VALUE assignment*)							UINT_TO_WORD(REAL_TO_UINT((1600)/0.05)),
(*ERROR is active*)										16#FEFE),
(*NOT AVAILABLE is active*)								16#FFFF),
(*Transmission is VALID*)								UINT_TO_WORD(REAL_TO_UINT((GVL.IOVD.X_I_Brk_Rsr.x + 1600)/0.05))),
		X_BYTE_0										=> _FB_CanTx_Message_464.X_Byte_2,
		X_BYTE_1										=> _FB_CanTx_Message_464.X_Byte_3);
{endregion}

{region " SIGNAL AREA : NAME->X_P_Mot_Cnv LENGTH->16 STARTBIT :32"}
_FB_UNPACK_WORD_TO_BYTE_9(
		X_WORD_0										:= 
(*SELECT 1 : Is data valid and range is not exceed?*)	SEL((GVL.IOVD.X_P_Mot_Cnv.v AND NOT GVL.IOVD.X_P_Mot_Cnv.RangeExcd),
(*SELECT 2 : Is NOT AVAILABLE ?*)						SEL(GVL.IOVD.X_P_Mot_Cnv.na,
(*SELECT 3 : Is ERROR active ?*)						SEL(GVL.IOVD.X_P_Mot_Cnv.e,
(*DEFAULT VALUE assignment*)							UINT_TO_WORD(REAL_TO_UINT((750)/0.025)),
(*ERROR is active*)										16#FEFE),
(*NOT AVAILABLE is active*)								16#FFFF),
(*Transmission is VALID*)								UINT_TO_WORD(REAL_TO_UINT((GVL.IOVD.X_P_Mot_Cnv.x + 750)/0.025))),
		X_BYTE_0										=> _FB_CanTx_Message_464.X_Byte_4,
		X_BYTE_1										=> _FB_CanTx_Message_464.X_Byte_5);
{endregion}

{region " SIGNAL AREA : NAME->X_P_Brk_Rsr LENGTH->16 STARTBIT :48"}
_FB_UNPACK_WORD_TO_BYTE_10(
		X_WORD_0										:= 
(*SELECT 1 : Is data valid and range is not exceed?*)	SEL((GVL.IOVD.X_P_Brk_Rsr.v AND NOT GVL.IOVD.X_P_Brk_Rsr.RangeExcd),
(*SELECT 2 : Is NOT AVAILABLE ?*)						SEL(GVL.IOVD.X_P_Brk_Rsr.na,
(*SELECT 3 : Is ERROR active ?*)						SEL(GVL.IOVD.X_P_Brk_Rsr.e,
(*DEFAULT VALUE assignment*)							UINT_TO_WORD(REAL_TO_UINT((750)/0.025)),
(*ERROR is active*)										16#FEFE),
(*NOT AVAILABLE is active*)								16#FFFF),
(*Transmission is VALID*)								UINT_TO_WORD(REAL_TO_UINT((GVL.IOVD.X_P_Brk_Rsr.x + 750)/0.025))),
		X_BYTE_0										=> _FB_CanTx_Message_464.X_Byte_6,
		X_BYTE_1										=> _FB_CanTx_Message_464.X_Byte_7);
{endregion}

_FB_CanTx_Message_464 (		C_Enable		:= GVL.IOVD.C_En_TCU_Cikis_Akim_Guc_0X464,
     						Obj_CAN			:= ADR(GVL.IC.Obj_CAN0),
     						X_MsgID			:= 16#464,
     						Tm_CycleTime	:= TIME#250MS,
     						N_Msg_Dlc		:= 8,
     						S_Extended		:= 0,
     						S_Sent_Ok   	=> GVL.IOVD.S_SentOk_TCU_Cikis_Akim_Guc_0X464);
{endregion}
//-----------------------------------------------------------------------------------------------------------------------------
//-----------------------------------------------------------------------------------------------------------------------------
{region " MESSAGE AREA :TCU_Tork_Hiz- ID:465"}

{region " SIGNAL AREA : NAME->X_M_Act LENGTH->16 STARTBIT :0"}
_FB_UNPACK_WORD_TO_BYTE_11 (
		X_WORD_0										:= 
(*SELECT 1 : Is data valid and range is not exceed?*)	SEL((GVL.IOVD.X_M_Act.v AND NOT GVL.IOVD.X_M_Act.RangeExcd),
(*SELECT 2 : Is NOT AVAILABLE ?*)						SEL(GVL.IOVD.X_M_Act.na,
(*SELECT 3 : Is ERROR active ?*)						SEL(GVL.IOVD.X_M_Act.e,
(*DEFAULT VALUE assignment*)							UINT_TO_WORD(REAL_TO_UINT((32766))),
(*ERROR is active*)										16#FEFE),
(*NOT AVAILABLE is active*)								16#FFFF),
(*Transmission is VALID*)								UINT_TO_WORD(REAL_TO_UINT((GVL.IOVD.X_M_Act.x + 32766)))),
		X_BYTE_0										=> _FB_CanTx_Message_465.X_Byte_0,
		X_BYTE_1										=> _FB_CanTx_Message_465.X_Byte_1);
{endregion}

{region " SIGNAL AREA : NAME->X_Spd_Act LENGTH->16 STARTBIT :16"}
_FB_UNPACK_WORD_TO_BYTE_12 (
		X_WORD_0										:= 
(*SELECT 1 : Is data valid and range is not exceed?*)	SEL((GVL.IOVD.X_Spd_Act.v AND NOT GVL.IOVD.X_Spd_Act.RangeExcd),
(*SELECT 2 : Is NOT AVAILABLE ?*)						SEL(GVL.IOVD.X_Spd_Act.na,
(*SELECT 3 : Is ERROR active ?*)						SEL(GVL.IOVD.X_Spd_Act.e,
(*DEFAULT VALUE assignment*)							UINT_TO_WORD(REAL_TO_UINT((32766))),
(*ERROR is active*)										16#FEFE),
(*NOT AVAILABLE is active*)								16#FFFF),
(*Transmission is VALID*)								UINT_TO_WORD(REAL_TO_UINT((GVL.IOVD.X_Spd_Act.x + 32766)))),
		X_BYTE_0										=> _FB_CanTx_Message_465.X_Byte_2,
		X_BYTE_1										=> _FB_CanTx_Message_465.X_Byte_3);
{endregion}

{region " SIGNAL AREA : NAME->X_Spd_Act_kmh LENGTH->16 STARTBIT :32"}
_FB_UNPACK_WORD_TO_BYTE_13 (
		X_WORD_0										:= 
(*SELECT 1 : Is data valid and range is not exceed?*)	SEL((GVL.IOVD.X_Spd_Act_kmh.v AND NOT GVL.IOVD.X_Spd_Act_kmh.RangeExcd),
(*SELECT 2 : Is NOT AVAILABLE ?*)						SEL(GVL.IOVD.X_Spd_Act_kmh.na,
(*SELECT 3 : Is ERROR active ?*)						SEL(GVL.IOVD.X_Spd_Act_kmh.e,
(*DEFAULT VALUE assignment*)							0,
(*ERROR is active*)										16#FEFE),
(*NOT AVAILABLE is active*)								16#FFFF),
(*Transmission is VALID*)								UINT_TO_WORD(REAL_TO_UINT((GVL.IOVD.X_Spd_Act_kmh.x)/0.01))),
		X_BYTE_0										=> _FB_CanTx_Message_465.X_Byte_4,
		X_BYTE_1										=> _FB_CanTx_Message_465.X_Byte_5);

{endregion}

_FB_CanTx_Message_465.X_Byte_6	:= 16#FF;
_FB_CanTx_Message_465.X_Byte_7	:= 16#FF;
	 
_FB_CanTx_Message_465 (		C_Enable		:= GVL.IOVD.C_En_TCU_Tork_Hiz_0X465,
     						Obj_CAN			:= ADR(GVL.IC.Obj_CAN0),
     						X_MsgID			:= 16#465,
     						Tm_CycleTime	:= TIME#250MS,
     						N_Msg_Dlc		:= 8,
     						S_Extended		:= 0,
     						S_Sent_Ok  	 	=> GVL.IOVD.S_SentOk_TCU_Tork_Hiz_0X465);
{endregion}
//-----------------------------------------------------------------------------------------------------------------------------
//-----------------------------------------------------------------------------------------------------------------------------
{region " MESSAGE AREA :TCU_Calisma_Suresi- ID:466"}

{region " SIGNAL AREA : NAME->N_Tm_Trol_Md LENGTH->32 STARTBIT :0"}
_FB_UNPACK_DWORD_TO_BYTE_0 (
		X_DWORD_0										:= 
(*SELECT 1 : Is data valid and range is not exceed?*)	SEL((GVL.IOVD.N_Tm_Trol_Md.v AND NOT GVL.IOVD.N_Tm_Trol_Md.RangeExcd),
(*SELECT 2 : Is NOT AVAILABLE ?*)						SEL(GVL.IOVD.N_Tm_Trol_Md.na,
(*SELECT 3 : Is ERROR active ?*)						SEL(GVL.IOVD.N_Tm_Trol_Md.e,
(*DEFAULT VALUE assignment*)							0,
(*ERROR is active*)										16#FEFEFEFE),
(*NOT AVAILABLE is active*)								16#FFFFFFFF),
(*Transmission is VALID*)								UDINT_TO_DWORD(GVL.IOVD.N_Tm_Trol_Md.x )),
		X_BYTE_0										=> _FB_CanTx_Message_466.X_Byte_0,
		X_BYTE_1										=> _FB_CanTx_Message_466.X_Byte_1,
		X_BYTE_2										=> _FB_CanTx_Message_466.X_Byte_2,
		X_BYTE_3										=> _FB_CanTx_Message_466.X_Byte_3);
{endregion}

{region " SIGNAL AREA : NAME->N_Tm_Bat_Md LENGTH->32 STARTBIT :32"}
_FB_UNPACK_DWORD_TO_BYTE_1 (
		X_DWORD_0										:= 
(*SELECT 1 : Is data valid and range is not exceed?*)	SEL((GVL.IOVD.N_Tm_Bat_Md.v AND NOT GVL.IOVD.N_Tm_Bat_Md.RangeExcd),
(*SELECT 2 : Is NOT AVAILABLE ?*)						SEL(GVL.IOVD.N_Tm_Bat_Md.na,
(*SELECT 3 : Is ERROR active ?*)						SEL(GVL.IOVD.N_Tm_Bat_Md.e,
(*DEFAULT VALUE assignment*)							0,
(*ERROR is active*)										16#FEFEFEFE),
(*NOT AVAILABLE is active*)								16#FFFFFFFF),
(*Transmission is VALID*)								UDINT_TO_DWORD(GVL.IOVD.N_Tm_Bat_Md.x )),
		X_BYTE_0										=> _FB_CanTx_Message_466.X_Byte_4,
		X_BYTE_1										=> _FB_CanTx_Message_466.X_Byte_5,
		X_BYTE_2										=> _FB_CanTx_Message_466.X_Byte_6,
		X_BYTE_3										=> _FB_CanTx_Message_466.X_Byte_7);
{endregion}

_FB_CanTx_Message_466 (		C_Enable		:= GVL.IOVD.C_En_TCU_Calisma_Suresi_0X466,
     						Obj_CAN			:= ADR(GVL.IC.Obj_CAN0),
     						X_MsgID			:= 16#466,
     						Tm_CycleTime	:= TIME#250MS,
     						N_Msg_Dlc		:= 8,
     						S_Extended		:= 0,
     						S_Sent_Ok   	=> GVL.IOVD.S_SentOk_TCU_Calisma_Suresi_0X466);
{endregion}
//-----------------------------------------------------------------------------------------------------------------------------
//-----------------------------------------------------------------------------------------------------------------------------
{region " MESSAGE AREA :TCU_Analog_2- ID:467"}

{region " SIGNAL AREA : NAME->X_U_Inv_HV LENGTH->16 STARTBIT :0"}
_FB_UNPACK_WORD_TO_BYTE_14 (
		X_WORD_0										:= 
(*SELECT 1 : Is data valid and range is not exceed?*)	SEL((GVL.IOVD.X_U_Inv_HV.v AND NOT GVL.IOVD.X_U_Inv_HV.RangeExcd),
(*SELECT 2 : Is NOT AVAILABLE ?*)						SEL(GVL.IOVD.X_U_Inv_HV.na,
(*SELECT 3 : Is ERROR active ?*)						SEL(GVL.IOVD.X_U_Inv_HV.e,
(*DEFAULT VALUE assignment*)							0,
(*ERROR is active*)										16#FEFE),
(*NOT AVAILABLE is active*)								16#FFFF),
(*Transmission is VALID*)								UINT_TO_WORD(REAL_TO_UINT((GVL.IOVD.X_U_Inv_HV.x)/0.025))),
		X_BYTE_0										=> _FB_CanTx_Message_467.X_Byte_0,
		X_BYTE_1										=> _FB_CanTx_Message_467.X_Byte_1);
{endregion}

{region " SIGNAL AREA : NAME->X_U_Cat_Ln LENGTH->16 STARTBIT :16"}
_FB_UNPACK_WORD_TO_BYTE_15 (
		X_WORD_0										:= 
(*SELECT 1 : Is data valid and range is not exceed?*)	SEL((GVL.IOVD.X_U_Cat_Ln.v AND NOT GVL.IOVD.X_U_Cat_Ln.RangeExcd),
(*SELECT 2 : Is NOT AVAILABLE ?*)						SEL(GVL.IOVD.X_U_Cat_Ln.na,
(*SELECT 3 : Is ERROR active ?*)						SEL(GVL.IOVD.X_U_Cat_Ln.e,
(*DEFAULT VALUE assignment*)							0,
(*ERROR is active*)										16#FEFE),
(*NOT AVAILABLE is active*)								16#FFFF),
(*Transmission is VALID*)								UINT_TO_WORD(REAL_TO_UINT((GVL.IOVD.X_U_Cat_Ln.x)/0.025))),
		X_BYTE_0										=> _FB_CanTx_Message_467.X_Byte_2,
		X_BYTE_1										=> _FB_CanTx_Message_467.X_Byte_3);
{endregion}

_FB_CanTx_Message_467.X_Byte_4:=16#FF;
_FB_CanTx_Message_467.X_Byte_5:=16#FF;
_FB_CanTx_Message_467.X_Byte_6:=16#FF;
_FB_CanTx_Message_467.X_Byte_7:=16#FF;
_FB_CanTx_Message_467(
     C_Enable:= GVL.IOVD.C_En_TCU_Analog_2_0X467,
     Obj_CAN:= ADR(GVL.IC.Obj_CAN0),
     X_MsgID:= 16#467,
     Tm_CycleTime:= TIME#250ms,
     N_Msg_Dlc:=8,
     S_Extended:= 0,
     S_Sent_Ok   => GVL.IOVD.S_SentOk_TCU_Analog_2_0X467);
{endregion}
//-----------------------------------------------------------------------------------------------------------------------------
//-----------------------------------------------------------------------------------------------------------------------------
{region " MESSAGE AREA :Yardimci_Konvertor_Durum- ID:480"}

{region " SIGNAL AREA : NAME->S_Aux_AC_Cnv_Rdy LENGTH->2 STARTBIT :0"}
_FB_CanTx_Message_Unpack_480.S_Bit_0		:= (GVL.IOVD.S_Aux_AC_Cnv_Rdy.x OR GVL.IOVD.S_Aux_AC_Cnv_Rdy.na) AND NOT GVL.IOVD.S_Aux_AC_Cnv_Rdy.e; 
_FB_CanTx_Message_Unpack_480.S_Bit_1		:= NOT GVL.IOVD.S_Aux_AC_Cnv_Rdy.v OR GVL.IOVD.S_Aux_AC_Cnv_Rdy.na OR GVL.IOVD.S_Aux_AC_Cnv_Rdy.e; 
{endregion}

{region " SIGNAL AREA : NAME->C_Aux_AC_Cnv_On LENGTH->2 STARTBIT :2"}
_FB_CanTx_Message_Unpack_480.S_Bit_2		:= (GVL.IOVD.C_Aux_AC_Cnv_On.x OR GVL.IOVD.C_Aux_AC_Cnv_On.na) AND NOT GVL.IOVD.C_Aux_AC_Cnv_On.e; 
_FB_CanTx_Message_Unpack_480.S_Bit_3		:= NOT GVL.IOVD.C_Aux_AC_Cnv_On.v OR GVL.IOVD.C_Aux_AC_Cnv_On.na OR GVL.IOVD.C_Aux_AC_Cnv_On.e; 
{endregion}

{region " SIGNAL AREA : NAME->S_Aux_AC_Cnv_On LENGTH->2 STARTBIT :4"}
_FB_CanTx_Message_Unpack_480.S_Bit_4		:= (GVL.IOVD.S_Aux_AC_Cnv_On.x OR GVL.IOVD.S_Aux_AC_Cnv_On.na) AND NOT GVL.IOVD.S_Aux_AC_Cnv_On.e; 
_FB_CanTx_Message_Unpack_480.S_Bit_5		:= NOT GVL.IOVD.S_Aux_AC_Cnv_On.v OR GVL.IOVD.S_Aux_AC_Cnv_On.na OR GVL.IOVD.S_Aux_AC_Cnv_On.e; 
{endregion}

{region " SIGNAL AREA : NAME->S_Aux_DC_24V_Cnv_Rdy LENGTH->2 STARTBIT :6"}
_FB_CanTx_Message_Unpack_480.S_Bit_6		:= (GVL.IOVD.S_Aux_DC_24V_Cnv_Rdy.x OR GVL.IOVD.S_Aux_DC_24V_Cnv_Rdy.na) AND NOT GVL.IOVD.S_Aux_DC_24V_Cnv_Rdy.e; 
_FB_CanTx_Message_Unpack_480.S_Bit_7		:= NOT GVL.IOVD.S_Aux_DC_24V_Cnv_Rdy.v OR GVL.IOVD.S_Aux_DC_24V_Cnv_Rdy.na OR GVL.IOVD.S_Aux_DC_24V_Cnv_Rdy.e; 
{endregion}

{region " SIGNAL AREA : NAME->C_Aux_DC_24V_Cnv_On LENGTH->2 STARTBIT :8"}
_FB_CanTx_Message_Unpack_480.S_Bit_8		:= (GVL.IOVD.C_Aux_DC_24V_Cnv_On.x OR GVL.IOVD.C_Aux_DC_24V_Cnv_On.na) AND NOT GVL.IOVD.C_Aux_DC_24V_Cnv_On.e; 
_FB_CanTx_Message_Unpack_480.S_Bit_9		:=  NOT GVL.IOVD.C_Aux_DC_24V_Cnv_On.v OR GVL.IOVD.C_Aux_DC_24V_Cnv_On.na OR GVL.IOVD.C_Aux_DC_24V_Cnv_On.e; 
{endregion}

{region " SIGNAL AREA : NAME->S_Aux_DC_24V_Cnv_On LENGTH->2 STARTBIT :10"}
_FB_CanTx_Message_Unpack_480.S_Bit_10		:= (GVL.IOVD.S_Aux_DC_24V_Cnv_On.x OR GVL.IOVD.S_Aux_DC_24V_Cnv_On.na) AND NOT GVL.IOVD.S_Aux_DC_24V_Cnv_On.e; 
_FB_CanTx_Message_Unpack_480.S_Bit_11		:= NOT GVL.IOVD.S_Aux_DC_24V_Cnv_On.v OR GVL.IOVD.S_Aux_DC_24V_Cnv_On.na OR GVL.IOVD.S_Aux_DC_24V_Cnv_On.e; 
{endregion}

{region " SIGNAL AREA : NAME->C_Aux_DC_Cnv_On LENGTH->2 STARTBIT :12"}
_FB_CanTx_Message_Unpack_480.S_Bit_12		:= (GVL.IOVD.C_Aux_DC_Cnv_On.x OR GVL.IOVD.C_Aux_DC_Cnv_On.na) AND NOT GVL.IOVD.C_Aux_DC_Cnv_On.e; 
_FB_CanTx_Message_Unpack_480.S_Bit_13		:= NOT GVL.IOVD.C_Aux_DC_Cnv_On.v OR GVL.IOVD.C_Aux_DC_Cnv_On.na OR GVL.IOVD.C_Aux_DC_Cnv_On.e; 
{endregion}

{region " SIGNAL AREA : NAME->S_Aux_DC_Cnv_On LENGTH->2 STARTBIT :14"}
_FB_CanTx_Message_Unpack_480.S_Bit_14		:= (GVL.IOVD.S_Aux_DC_Cnv_On.x OR GVL.IOVD.S_Aux_DC_Cnv_On.na) AND NOT GVL.IOVD.S_Aux_DC_Cnv_On.e; 
_FB_CanTx_Message_Unpack_480.S_Bit_15		:= NOT GVL.IOVD.S_Aux_DC_Cnv_On.v OR GVL.IOVD.S_Aux_DC_Cnv_On.na OR GVL.IOVD.S_Aux_DC_Cnv_On.e; 
{endregion}

{region " SIGNAL AREA : NAME->C_Bat_Chrg_DC_Cnv_On LENGTH->2 STARTBIT :16"}
_FB_CanTx_Message_Unpack_480.S_Bit_16		:= (GVL.IOVD.C_Bat_Chrg_DC_Cnv_On.x OR GVL.IOVD.C_Bat_Chrg_DC_Cnv_On.na) AND NOT GVL.IOVD.C_Bat_Chrg_DC_Cnv_On.e; 
_FB_CanTx_Message_Unpack_480.S_Bit_17		:= NOT GVL.IOVD.C_Bat_Chrg_DC_Cnv_On.v OR GVL.IOVD.C_Bat_Chrg_DC_Cnv_On.na OR GVL.IOVD.C_Bat_Chrg_DC_Cnv_On.e; 
{endregion}

{region " SIGNAL AREA : NAME->S_Bat_Chrg_DC_Cnv_On LENGTH->2 STARTBIT :18"}
_FB_CanTx_Message_Unpack_480.S_Bit_18		:= (GVL.IOVD.S_Bat_Chrg_DC_Cnv_On.x OR GVL.IOVD.S_Bat_Chrg_DC_Cnv_On.na) AND NOT GVL.IOVD.S_Bat_Chrg_DC_Cnv_On.e; 
_FB_CanTx_Message_Unpack_480.S_Bit_19		:= NOT GVL.IOVD.S_Bat_Chrg_DC_Cnv_On.v OR GVL.IOVD.S_Bat_Chrg_DC_Cnv_On.na OR GVL.IOVD.S_Bat_Chrg_DC_Cnv_On.e; 
{endregion}

{region " SIGNAL AREA : NAME->C_Aux_DC_Ct_1_On LENGTH->2 STARTBIT :20"}
_FB_CanTx_Message_Unpack_480.S_Bit_20		:= (GVL.IOVD.C_Aux_DC_Ct_1_On.x OR GVL.IOVD.C_Aux_DC_Ct_1_On.na) AND NOT GVL.IOVD.C_Aux_DC_Ct_1_On.e; 
_FB_CanTx_Message_Unpack_480.S_Bit_21		:= NOT GVL.IOVD.C_Aux_DC_Ct_1_On.v OR GVL.IOVD.C_Aux_DC_Ct_1_On.na OR GVL.IOVD.C_Aux_DC_Ct_1_On.e; 
{endregion}

{region " SIGNAL AREA : NAME->C_Aux_DC_Ct_2_On LENGTH->2 STARTBIT :22"}
_FB_CanTx_Message_Unpack_480.S_Bit_22		:= (GVL.IOVD.C_Aux_DC_Ct_2_On.x OR GVL.IOVD.C_Aux_DC_Ct_2_On.na) AND NOT GVL.IOVD.C_Aux_DC_Ct_2_On.e; 
_FB_CanTx_Message_Unpack_480.S_Bit_23		:= NOT GVL.IOVD.C_Aux_DC_Ct_2_On.v OR GVL.IOVD.C_Aux_DC_Ct_2_On.na OR GVL.IOVD.C_Aux_DC_Ct_2_On.e; 
{endregion}

{region " SIGNAL AREA : NAME->C_Aux_DC_Ct_3_On LENGTH->2 STARTBIT :24"}
_FB_CanTx_Message_Unpack_480.S_Bit_24		:= (GVL.IOVD.C_Aux_DC_Ct_3_On.x OR GVL.IOVD.C_Aux_DC_Ct_3_On.na) AND NOT GVL.IOVD.C_Aux_DC_Ct_3_On.e; 
_FB_CanTx_Message_Unpack_480.S_Bit_25		:= NOT GVL.IOVD.C_Aux_DC_Ct_3_On.v OR GVL.IOVD.C_Aux_DC_Ct_3_On.na OR GVL.IOVD.C_Aux_DC_Ct_3_On.e; 
{endregion}

{region " SIGNAL AREA : NAME->S_Aux_DC_Ct_1_Actv LENGTH->2 STARTBIT :26"}
_FB_CanTx_Message_Unpack_480.S_Bit_26		:= (GVL.IOVD.S_Aux_DC_Ct_1_Actv.x OR GVL.IOVD.S_Aux_DC_Ct_1_Actv.na) AND NOT GVL.IOVD.S_Aux_DC_Ct_1_Actv.e; 
_FB_CanTx_Message_Unpack_480.S_Bit_27		:= NOT GVL.IOVD.S_Aux_DC_Ct_1_Actv.v OR GVL.IOVD.S_Aux_DC_Ct_1_Actv.na OR GVL.IOVD.S_Aux_DC_Ct_1_Actv.e; 
{endregion}

{region " SIGNAL AREA : NAME->S_Aux_DC_Ct_2_Actv LENGTH->2 STARTBIT :28"}
_FB_CanTx_Message_Unpack_480.S_Bit_28		:= (GVL.IOVD.S_Aux_DC_Ct_2_Actv.x OR GVL.IOVD.S_Aux_DC_Ct_2_Actv.na) AND NOT GVL.IOVD.S_Aux_DC_Ct_2_Actv.e; 
_FB_CanTx_Message_Unpack_480.S_Bit_29		:=	NOT GVL.IOVD.S_Aux_DC_Ct_2_Actv.v OR GVL.IOVD.S_Aux_DC_Ct_2_Actv.na OR GVL.IOVD.S_Aux_DC_Ct_2_Actv.e; 
{endregion}

{region " SIGNAL AREA : NAME->S_Aux_DC_Ct_3_Actv LENGTH->2 STARTBIT :30"}
_FB_CanTx_Message_Unpack_480.S_Bit_30		:= (GVL.IOVD.S_Aux_DC_Ct_3_Actv.x OR GVL.IOVD.S_Aux_DC_Ct_3_Actv.na) AND NOT GVL.IOVD.S_Aux_DC_Ct_3_Actv.e; 
_FB_CanTx_Message_Unpack_480.S_Bit_31		:= NOT GVL.IOVD.S_Aux_DC_Ct_3_Actv.v OR GVL.IOVD.S_Aux_DC_Ct_3_Actv.na OR GVL.IOVD.S_Aux_DC_Ct_3_Actv.e; 
{endregion}

{region " SIGNAL AREA : NAME->Z_Bccu_Stat LENGTH->8 STARTBIT :32"}
_FB_CanTx_Message_Unpack_480.X_Byte_4					:=
(*SELECT 1 : Is data valid and range is not exceed?*)	SEL((GVL.IOVD.Z_Bccu_Stat.v AND NOT GVL.IOVD.Z_Bccu_Stat.RangeExcd),
(*SELECT 2 : Is NOT AVAILABLE ?*)						SEL(GVL.IOVD.Z_Bccu_Stat.na,
(*SELECT 3 : Is ERROR active ?*)						SEL(GVL.IOVD.Z_Bccu_Stat.e,
(*DEFAULT VALUE assignment*)							0,
(*ERROR is active*)										16#FE),
(*NOT AVAILABLE is active*)								16#FF),
(*Transmission is VALID*)								GVL.IOVD.Z_Bccu_Stat.x);
{endregion}

{region " SIGNAL AREA : NAME->Z_Tcu_Stat LENGTH->8 STARTBIT :32"}
_FB_CanTx_Message_Unpack_480.X_Byte_5					:=
(*SELECT 1 : Is data valid and range is not exceed?*)	SEL((GVL.IOVD.Z_Tcu_Stat.v AND NOT GVL.IOVD.Z_Tcu_Stat.RangeExcd),
(*SELECT 2 : Is NOT AVAILABLE ?*)						SEL(GVL.IOVD.Z_Tcu_Stat.na,
(*SELECT 3 : Is ERROR active ?*)						SEL(GVL.IOVD.Z_Tcu_Stat.e,
(*DEFAULT VALUE assignment*)							0,
(*ERROR is active*)										16#FE),
(*NOT AVAILABLE is active*)								16#FF),
(*Transmission is VALID*)								GVL.IOVD.Z_Tcu_Stat.x);
{endregion}	

{region " SIGNAL AREA : NAME->Z_Apu_Stat LENGTH->8 STARTBIT :32"}
_FB_CanTx_Message_Unpack_480.X_Byte_6					:=
(*SELECT 1 : Is data valid and range is not exceed?*)	SEL((GVL.IOVD.Z_Apu_Stat.v AND NOT GVL.IOVD.Z_Apu_Stat.RangeExcd),
(*SELECT 2 : Is NOT AVAILABLE ?*)						SEL(GVL.IOVD.Z_Apu_Stat.na,
(*SELECT 3 : Is ERROR active ?*)						SEL(GVL.IOVD.Z_Apu_Stat.e,
(*DEFAULT VALUE assignment*)							0,
(*ERROR is active*)										16#FE),
(*NOT AVAILABLE is active*)								16#FF),
(*Transmission is VALID*)								GVL.IOVD.Z_Apu_Stat.x);
{endregion}			   

_FB_CanTx_Message_Unpack_480.X_Byte_7	:= 16#FF;

_FB_CanTx_Message_Unpack_480 (		C_Enable		:= GVL.IOVD.C_En_Yardimci_Konvertor_Durum_0X480,
     								Obj_CAN			:= ADR(GVL.IC.Obj_CAN0),
     								X_MsgID			:= 16#480,
     								Tm_CycleTime	:= TIME#250MS,
     								N_Msg_Dlc		:= 8,
     								S_Extended		:= 0,
     								S_Sent_Ok   	=> GVL.IOVD.S_SentOk_Yardimci_Konvertor_Durum_0X480);
{endregion}
//-----------------------------------------------------------------------------------------------------------------------------
//-----------------------------------------------------------------------------------------------------------------------------
{region " MESSAGE AREA :Yardimci_Konvertor_Akim- ID:481"}

{region " SIGNAL AREA : NAME->X_I_Out_Aux_DC_Cnv LENGTH->16 STARTBIT :0"}
_FB_UNPACK_WORD_TO_BYTE_16 (
		X_WORD_0										:= 
(*SELECT 1 : Is data valid and range is not exceed?*)	SEL((GVL.IOVD.X_I_Out_Aux_DC_Cnv.v AND NOT GVL.IOVD.X_I_Out_Aux_DC_Cnv.RangeExcd),
(*SELECT 2 : Is NOT AVAILABLE ?*)						SEL(GVL.IOVD.X_I_Out_Aux_DC_Cnv.na,
(*SELECT 3 : Is ERROR active ?*)						SEL(GVL.IOVD.X_I_Out_Aux_DC_Cnv.e,
(*DEFAULT VALUE assignment*)							0,
(*ERROR is active*)										16#FEFE),
(*NOT AVAILABLE is active*)								16#FFFF),
(*Transmission is VALID*)								UINT_TO_WORD(REAL_TO_UINT((GVL.IOVD.X_I_Out_Aux_DC_Cnv.x)/0.1))),
		X_BYTE_0										=> _FB_CanTx_Message_Unpack_481.X_Byte_0,
		X_BYTE_1										=> _FB_CanTx_Message_Unpack_481.X_Byte_1);
{endregion}

{region " SIGNAL AREA : NAME->X_I_Out_Aux_AC_Cnv LENGTH->16 STARTBIT :16"}
_FB_UNPACK_WORD_TO_BYTE_17 (
		X_WORD_0										:= 
(*SELECT 1 : Is data valid and range is not exceed?*)	SEL((GVL.IOVD.X_I_Out_Aux_AC_Cnv.v AND NOT GVL.IOVD.X_I_Out_Aux_AC_Cnv.RangeExcd),
(*SELECT 2 : Is NOT AVAILABLE ?*)						SEL(GVL.IOVD.X_I_Out_Aux_AC_Cnv.na,
(*SELECT 3 : Is ERROR active ?*)						SEL(GVL.IOVD.X_I_Out_Aux_AC_Cnv.e,
(*DEFAULT VALUE assignment*)							0,
(*ERROR is active*)										16#FEFE),
(*NOT AVAILABLE is active*)								16#FFFF),
(*Transmission is VALID*)								UINT_TO_WORD(REAL_TO_UINT((GVL.IOVD.X_I_Out_Aux_AC_Cnv.x)/0.1))),
		X_BYTE_0										=> _FB_CanTx_Message_Unpack_481.X_Byte_2,
		X_BYTE_1										=> _FB_CanTx_Message_Unpack_481.X_Byte_3);
{endregion}

{region " SIGNAL AREA : NAME->X_I_Out_Aux_DC_24V_Cnv LENGTH->16 STARTBIT :32"}
_FB_UNPACK_WORD_TO_BYTE_18 (
		X_WORD_0										:= 
(*SELECT 1 : Is data valid and range is not exceed?*)	SEL((GVL.IOVD.X_I_Out_Aux_DC_24V_Cnv.v AND NOT GVL.IOVD.X_I_Out_Aux_DC_24V_Cnv.RangeExcd),
(*SELECT 2 : Is NOT AVAILABLE ?*)						SEL(GVL.IOVD.X_I_Out_Aux_DC_24V_Cnv.na,
(*SELECT 3 : Is ERROR active ?*)						SEL(GVL.IOVD.X_I_Out_Aux_DC_24V_Cnv.e,
(*DEFAULT VALUE assignment*)							UINT_TO_WORD(REAL_TO_UINT((750)/0.025)),
(*ERROR is active*)										16#FEFE),
(*NOT AVAILABLE is active*)								16#FFFF),
(*Transmission is VALID*)								UINT_TO_WORD(REAL_TO_UINT((GVL.IOVD.X_I_Out_Aux_DC_24V_Cnv.x + 750)/0.025))),
		X_BYTE_0										=> _FB_CanTx_Message_Unpack_481.X_Byte_4,
		X_BYTE_1										=> _FB_CanTx_Message_Unpack_481.X_Byte_5);
{endregion}

{region " SIGNAL AREA : NAME->X_I_In_Aux_DC_24V_Cnv LENGTH->16 STARTBIT :48"}
_FB_UNPACK_WORD_TO_BYTE_19 (
		X_WORD_0										:= 
(*SELECT 1 : Is data valid and range is not exceed?*)	SEL((GVL.IOVD.X_I_In_Aux_DC_24V_Cnv.v AND NOT GVL.IOVD.X_I_In_Aux_DC_24V_Cnv.RangeExcd),
(*SELECT 2 : Is NOT AVAILABLE ?*)						SEL(GVL.IOVD.X_I_In_Aux_DC_24V_Cnv.na,
(*SELECT 3 : Is ERROR active ?*)						SEL(GVL.IOVD.X_I_In_Aux_DC_24V_Cnv.e,
(*DEFAULT VALUE assignment*)							0,
(*ERROR is active*)										16#FEFE),
(*NOT AVAILABLE is active*)								16#FFFF),
(*Transmission is VALID*)								UINT_TO_WORD(REAL_TO_UINT((GVL.IOVD.X_I_In_Aux_DC_24V_Cnv.x)/0.1))),
		X_BYTE_0										=> _FB_CanTx_Message_Unpack_481.X_Byte_6,
		X_BYTE_1										=> _FB_CanTx_Message_Unpack_481.X_Byte_7);
{endregion}

_FB_CanTx_Message_Unpack_481(
     C_Enable:= GVL.IOVD.C_En_Yardimci_Konvertor_Akim_0X481,
     Obj_CAN:= ADR(GVL.IC.Obj_CAN0),
     X_MsgID:= 16#481,
     Tm_CycleTime:= TIME#250ms,
     N_Msg_Dlc:=8,
     S_Extended:= 0,
     S_Sent_Ok   => GVL.IOVD.S_SentOk_Yardimci_Konvertor_Akim_0X481);
{endregion}
//-----------------------------------------------------------------------------------------------------------------------------
//-----------------------------------------------------------------------------------------------------------------------------
{region " MESSAGE AREA :Yardimci_Konvertor_Guc- ID:482"}

{region " SIGNAL AREA : NAME->X_U_Out_24V_Bat LENGTH->16 STARTBIT :0"}
_FB_UNPACK_WORD_TO_BYTE_20 (
		X_WORD_0										:= 
(*SELECT 1 : Is data valid and range is not exceed?*)	SEL((GVL.IOVD.X_U_Out_24V_Bat.v AND NOT GVL.IOVD.X_U_Out_24V_Bat.RangeExcd),
(*SELECT 2 : Is NOT AVAILABLE ?*)						SEL(GVL.IOVD.X_U_Out_24V_Bat.na,
(*SELECT 3 : Is ERROR active ?*)						SEL(GVL.IOVD.X_U_Out_24V_Bat.e,
(*DEFAULT VALUE assignment*)							0,
(*ERROR is active*)										16#FEFE),
(*NOT AVAILABLE is active*)								16#FFFF),
(*Transmission is VALID*)								UINT_TO_WORD(REAL_TO_UINT((GVL.IOVD.X_U_Out_24V_Bat.x)/0.01))),
		X_BYTE_0										=> _FB_CanTx_Message_Unpack_482.X_Byte_0,
		X_BYTE_1										=> _FB_CanTx_Message_Unpack_482.X_Byte_1);
{endregion}

{region " SIGNAL AREA : NAME->X_P_Out_Aux_DC_Cnv LENGTH->16 STARTBIT :16"}
_FB_UNPACK_WORD_TO_BYTE_21 (
		X_WORD_0										:= 
(*SELECT 1 : Is data valid and range is not exceed?*)	SEL((GVL.IOVD.X_P_Out_Aux_DC_Cnv.v AND NOT GVL.IOVD.X_P_Out_Aux_DC_Cnv.RangeExcd),
(*SELECT 2 : Is NOT AVAILABLE ?*)						SEL(GVL.IOVD.X_P_Out_Aux_DC_Cnv.na,
(*SELECT 3 : Is ERROR active ?*)						SEL(GVL.IOVD.X_P_Out_Aux_DC_Cnv.e,
(*DEFAULT VALUE assignment*)							UINT_TO_WORD(REAL_TO_UINT((750)/0.025)),
(*ERROR is active*)										16#FEFE),
(*NOT AVAILABLE is active*)								16#FFFF),
(*Transmission is VALID*)								UINT_TO_WORD(REAL_TO_UINT((GVL.IOVD.X_P_Out_Aux_DC_Cnv.x + 750)/0.025))),
		X_BYTE_0										=> _FB_CanTx_Message_Unpack_482.X_Byte_2,
		X_BYTE_1										=> _FB_CanTx_Message_Unpack_482.X_Byte_3);
{endregion}

{region " SIGNAL AREA : NAME->X_P_Out_Aux_AC_Cnv LENGTH->16 STARTBIT :32"}
_FB_UNPACK_WORD_TO_BYTE_22 (
		X_WORD_0										:= 
(*SELECT 1 : Is data valid and range is not exceed?*)	SEL((GVL.IOVD.X_P_Out_Aux_AC_Cnv.v AND NOT GVL.IOVD.X_P_Out_Aux_AC_Cnv.RangeExcd),
(*SELECT 2 : Is NOT AVAILABLE ?*)						SEL(GVL.IOVD.X_P_Out_Aux_AC_Cnv.na,
(*SELECT 3 : Is ERROR active ?*)						SEL(GVL.IOVD.X_P_Out_Aux_AC_Cnv.e,
(*DEFAULT VALUE assignment*)							UINT_TO_WORD(REAL_TO_UINT((750)/0.025)),
(*ERROR is active*)										16#FEFE),
(*NOT AVAILABLE is active*)								16#FFFF),
(*Transmission is VALID*)								UINT_TO_WORD(REAL_TO_UINT((GVL.IOVD.X_P_Out_Aux_AC_Cnv.x + 750)/0.025))),
		X_BYTE_0										=> _FB_CanTx_Message_Unpack_482.X_Byte_4,
		X_BYTE_1										=> _FB_CanTx_Message_Unpack_482.X_Byte_5);

{endregion}

{region " SIGNAL AREA : NAME->X_P_Out_Aux_DC_24V_Cnv LENGTH->16 STARTBIT :48"}
_FB_UNPACK_WORD_TO_BYTE_23 (
		X_WORD_0										:= 
(*SELECT 1 : Is data valid and range is not exceed?*)	SEL((GVL.IOVD.X_P_Out_Aux_DC_24V_Cnv.v AND NOT GVL.IOVD.X_P_Out_Aux_DC_24V_Cnv.RangeExcd),
(*SELECT 2 : Is NOT AVAILABLE ?*)						SEL(GVL.IOVD.X_P_Out_Aux_DC_24V_Cnv.na,
(*SELECT 3 : Is ERROR active ?*)						SEL(GVL.IOVD.X_P_Out_Aux_DC_24V_Cnv.e,
(*DEFAULT VALUE assignment*)							UINT_TO_WORD(REAL_TO_UINT((750)/0.025)),
(*ERROR is active*)										16#FEFE),
(*NOT AVAILABLE is active*)								16#FFFF),
(*Transmission is VALID*)								UINT_TO_WORD(REAL_TO_UINT((GVL.IOVD.X_P_Out_Aux_DC_24V_Cnv.x + 750)/0.025))),
		X_BYTE_0										=> _FB_CanTx_Message_Unpack_482.X_Byte_6,
		X_BYTE_1										=> _FB_CanTx_Message_Unpack_482.X_Byte_7);
{endregion}

_FB_CanTx_Message_Unpack_482 (		C_Enable		:= GVL.IOVD.C_En_Yardimci_Konvertor_Guc_0X482,
     								Obj_CAN			:= ADR(GVL.IC.Obj_CAN0),
     								X_MsgID			:= 16#482,
     								Tm_CycleTime	:= TIME#250MS,
     								N_Msg_Dlc		:= 8,
     								S_Extended		:= 0,
     								S_Sent_Ok   	=> GVL.IOVD.S_SentOk_Yardimci_Konvertor_Guc_0X482);
{endregion}
//-----------------------------------------------------------------------------------------------------------------------------
//-----------------------------------------------------------------------------------------------------------------------------
{region " MESSAGE AREA :Batarya_Sarj_Konvertor- ID:483"}

{region " SIGNAL AREA : NAME->X_P_Bat_Chrg_DC_Cnv LENGTH->16 STARTBIT :0"}
_FB_UNPACK_WORD_TO_BYTE_26 (
		X_WORD_0										:= 
(*SELECT 1 : Is data valid and range is not exceed?*)	SEL((GVL.IOVD.X_P_Bat_Chrg_DC_Cnv.v AND NOT GVL.IOVD.X_P_Bat_Chrg_DC_Cnv.RangeExcd),
(*SELECT 2 : Is NOT AVAILABLE ?*)						SEL(GVL.IOVD.X_P_Bat_Chrg_DC_Cnv.na,
(*SELECT 3 : Is ERROR active ?*)						SEL(GVL.IOVD.X_P_Bat_Chrg_DC_Cnv.e,
(*DEFAULT VALUE assignment*)							0,
(*ERROR is active*)										16#FEFE),
(*NOT AVAILABLE is active*)								16#FFFF),
(*Transmission is VALID*)								UINT_TO_WORD(REAL_TO_UINT((GVL.IOVD.X_P_Bat_Chrg_DC_Cnv.x + 3276.6)/0.1))),
		X_BYTE_0										=> _FB_CanTx_Message_Unpack_483.X_Byte_0,
		X_BYTE_1										=> _FB_CanTx_Message_Unpack_483.X_Byte_1);
{endregion}

{region " SIGNAL AREA : NAME->X_I_Out_Aux_Bat_Chrg_DC_Cnv LENGTH->16 STARTBIT :16"}
_FB_UNPACK_WORD_TO_BYTE_27 (
		X_WORD_0										:= 
(*SELECT 1 : Is data valid and range is not exceed?*)	SEL((GVL.IOVD.X_I_Out_Aux_Bat_Chrg_DC_Cnv.v AND NOT GVL.IOVD.X_I_Out_Aux_Bat_Chrg_DC_Cnv.RangeExcd),
(*SELECT 2 : Is NOT AVAILABLE ?*)						SEL(GVL.IOVD.X_I_Out_Aux_Bat_Chrg_DC_Cnv.na,
(*SELECT 3 : Is ERROR active ?*)						SEL(GVL.IOVD.X_I_Out_Aux_Bat_Chrg_DC_Cnv.e,
(*DEFAULT VALUE assignment*)							UINT_TO_WORD(REAL_TO_UINT((1600)/0.05)),
(*ERROR is active*)										16#FEFE),
(*NOT AVAILABLE is active*)								16#FFFF),
(*Transmission is VALID*)								UINT_TO_WORD(REAL_TO_UINT((GVL.IOVD.X_I_Out_Aux_Bat_Chrg_DC_Cnv.x + 1600)/0.05))),
		X_BYTE_0										=> _FB_CanTx_Message_Unpack_483.X_Byte_2,
		X_BYTE_1										=> _FB_CanTx_Message_Unpack_483.X_Byte_3);
{endregion}

_FB_CanTx_Message_Unpack_483.X_Byte_4		:= 16#FF;
_FB_CanTx_Message_Unpack_483.X_Byte_5		:= 16#FF;
_FB_CanTx_Message_Unpack_483.X_Byte_6		:= 16#FF;
_FB_CanTx_Message_Unpack_483.X_Byte_7		:= 16#FF; 

_FB_CanTx_Message_Unpack_483 (		C_Enable		:= GVL.IOVD.C_En_Batarya_Sarj_Konvertor_Analog_0X483,
     								Obj_CAN			:= ADR(GVL.IC.Obj_CAN0),
     								X_MsgID			:= 16#483,
     								Tm_CycleTime	:= TIME#250MS,
     								N_Msg_Dlc		:= 8,
     								S_Extended		:= 0,
     								S_Sent_Ok   	=> GVL.IOVD.S_SentOk_Batarya_Konvertor_Analog_0X483);
{endregion}

{region " MESSAGE AREA :Yardimci_Konvertor_Sicaklik- ID:484"}

{region " SIGNAL AREA : NAME->X_T_Aux_AC_Cnv LENGTH->8 STARTBIT :0"}
_FB_CanTx_Message_Unpack_484.X_Byte_0					:=
(*SELECT 1 : Is data valid and range is not exceed?*)	SEL((GVL.IOVD.X_T_Aux_AC_Cnv.v AND NOT GVL.IOVD.X_T_Aux_AC_Cnv.RangeExcd),
(*SELECT 2 : Is NOT AVAILABLE ?*)						SEL(GVL.IOVD.X_T_Aux_AC_Cnv.na,
(*SELECT 3 : Is ERROR active ?*)						SEL(GVL.IOVD.X_T_Aux_AC_Cnv.e,
(*DEFAULT VALUE assignment*)							USINT_TO_BYTE(REAL_TO_USINT((40))),
(*ERROR is active*)										16#FE),
(*NOT AVAILABLE is active*)								16#FF),
(*Transmission is VALID*)								USINT_TO_BYTE(REAL_TO_USINT((GVL.IOVD.X_T_Aux_AC_Cnv.x + 40))));
{endregion}

{region " SIGNAL AREA : NAME->X_T_Aux_DC_24V_Cnv LENGTH->8 STARTBIT :8"}
_FB_CanTx_Message_Unpack_484.X_Byte_1					:=
(*SELECT 1 : Is data valid and range is not exceed?*)	SEL((GVL.IOVD.X_T_Aux_DC_24V_Cnv.v AND NOT GVL.IOVD.X_T_Aux_DC_24V_Cnv.RangeExcd),
(*SELECT 2 : Is NOT AVAILABLE ?*)						SEL(GVL.IOVD.X_T_Aux_DC_24V_Cnv.na,
(*SELECT 3 : Is ERROR active ?*)						SEL(GVL.IOVD.X_T_Aux_DC_24V_Cnv.e,
(*DEFAULT VALUE assignment*)							USINT_TO_BYTE(REAL_TO_USINT((40))),
(*ERROR is active*)										16#FE),
(*NOT AVAILABLE is active*)								16#FF),
(*Transmission is VALID*)								USINT_TO_BYTE(REAL_TO_USINT((GVL.IOVD.X_T_Aux_DC_24V_Cnv.x + 40))));
{endregion}

{region " SIGNAL AREA : NAME->X_T_Aux_DC_Cnv LENGTH->8 STARTBIT :16"}
_FB_CanTx_Message_Unpack_484.X_Byte_2					:=
(*SELECT 1 : Is data valid and range is not exceed?*)	SEL((GVL.IOVD.X_T_Aux_DC_Cnv.v AND NOT GVL.IOVD.X_T_Aux_DC_Cnv.RangeExcd),
(*SELECT 2 : Is NOT AVAILABLE ?*)						SEL(GVL.IOVD.X_T_Aux_DC_Cnv.na,
(*SELECT 3 : Is ERROR active ?*)						SEL(GVL.IOVD.X_T_Aux_DC_Cnv.e,
(*DEFAULT VALUE assignment*)							USINT_TO_BYTE(REAL_TO_USINT((40))),
(*ERROR is active*)										16#FE),
(*NOT AVAILABLE is active*)								16#FF),
(*Transmission is VALID*)								USINT_TO_BYTE(REAL_TO_USINT((GVL.IOVD.X_T_Aux_DC_Cnv.x + 40))));
{endregion}

{region " SIGNAL AREA : NAME->X_T_Bat_Chrg_DC_Cnv LENGTH->8 STARTBIT :24"}
_FB_CanTx_Message_Unpack_484.X_Byte_3					:=
(*SELECT 1 : Is data valid and range is not exceed?*)	SEL((GVL.IOVD.X_T_Bat_Chrg_DC_Cnv.v AND NOT GVL.IOVD.X_T_Bat_Chrg_DC_Cnv.RangeExcd),
(*SELECT 2 : Is NOT AVAILABLE ?*)						SEL(GVL.IOVD.X_T_Bat_Chrg_DC_Cnv.na,
(*SELECT 3 : Is ERROR active ?*)						SEL(GVL.IOVD.X_T_Bat_Chrg_DC_Cnv.e,
(*DEFAULT VALUE assignment*)							USINT_TO_BYTE(REAL_TO_USINT((40))),
(*ERROR is active*)										16#FE),
(*NOT AVAILABLE is active*)								16#FF),
(*Transmission is VALID*)								USINT_TO_BYTE(REAL_TO_USINT((GVL.IOVD.X_T_Bat_Chrg_DC_Cnv.x + 40))));
{endregion}

_FB_CanTx_Message_Unpack_484.X_Byte_4	:= 16#FF;
_FB_CanTx_Message_Unpack_484.X_Byte_5	:= 16#FF;
_FB_CanTx_Message_Unpack_484.X_Byte_6	:= 16#FF;
_FB_CanTx_Message_Unpack_484.X_Byte_7	:= 16#FF;
	 
_FB_CanTx_Message_Unpack_484 (		C_Enable		:= GVL.IOVD.C_En_Yardimci_Konvertor_Sicaklik_0X484,
     								Obj_CAN			:= ADR(GVL.IC.Obj_CAN0),
     								X_MsgID			:= 16#484,
     								Tm_CycleTime	:= TIME#250MS,
     								N_Msg_Dlc		:= 8,
     								S_Extended		:= 0,
     								S_Sent_Ok   	=> GVL.IOVD.S_SentOk_Yardimci_Konvertor_Sicaklik_0X484);
{endregion}
//-----------------------------------------------------------------------------------------------------------------------------
//-----------------------------------------------------------------------------------------------------------------------------

{region " MESSAGE AREA :Isolation_Status - ID:485"}

{region " SIGNAL AREA : NAME->Z_Insu_Dev LENGTH->4 STARTBIT :0"}
_FB_UNPACK_BYTE_TO_8BITS_2(
		S_Bit_0=> _FB_CanTx_Message_Unpack_485.S_Bit_0,
		S_Bit_1=> _FB_CanTx_Message_Unpack_485.S_Bit_1,
		S_Bit_2=> _FB_CanTx_Message_Unpack_485.S_Bit_2,
		S_Bit_3=> _FB_CanTx_Message_Unpack_485.S_Bit_3,
		X_BYTE_0:=
(*SELECT 1 : Is data valid and range is not exceed?*)	SEL((GVL.IOVD.Z_Insu_Dev.v AND NOT GVL.IOVD.Z_Insu_Dev.RangeExcd),
(*SELECT 2 : Is NOT AVAILABLE ?*)						SEL(GVL.IOVD.Z_Insu_Dev.na,
(*SELECT 3 : Is ERROR active ?*)						SEL(GVL.IOVD.Z_Insu_Dev.e,
(*DEFAULT VALUE assignment*)							0,
(*ERROR is active*)										16#E),
(*NOT AVAILABLE is active*)								16#F),
(*Transmission is VALID*)								GVL.IOVD.Z_Insu_Dev.x));
{endregion}

{region " SIGNAL AREA : NAME->S_ER_Insu_Dev_Not_Conn LENGTH->1 STARTBIT :4"}
_FB_CanTx_Message_Unpack_485.S_Bit_4		:= GVL.IOVD.S_ER_Insu_Dev_Not_Conn.x AND GVL.IOVD.S_ER_Insu_Dev_Not_Conn.v;
{endregion}

{region " SIGNAL AREA : NAME->Z_Man_Insu_Tst LENGTH->8 STARTBIT :8"}
_FB_CanTx_Message_Unpack_485.X_Byte_1:=					SEL((GVL.IOVD.Z_Man_Insu_Tst.v AND NOT GVL.IOVD.Z_Man_Insu_Tst.RangeExcd),
(*SELECT 2 : Is NOT AVAILABLE ?*)						SEL(GVL.IOVD.Z_Man_Insu_Tst.na,
(*SELECT 3 : Is ERROR active ?*)						SEL(GVL.IOVD.Z_Man_Insu_Tst.e,
(*DEFAULT VALUE assignment*)							0,
(*ERROR is active*)										16#FE),
(*NOT AVAILABLE is active*)								16#FF),
(*Transmission is VALID*)								USINT_TO_BYTE(REAL_TO_USINT((GVL.IOVD.Z_Man_Insu_Tst.x))));
{endregion}

{region " SIGNAL AREA : NAME->Z_Semi_Aut_Insu_Tst LENGTH->8 STARTBIT :16"}
_FB_CanTx_Message_Unpack_485.X_Byte_2:=					SEL((GVL.IOVD.Z_Semi_Aut_Insu_Tst.v AND NOT GVL.IOVD.Z_Semi_Aut_Insu_Tst.RangeExcd),
(*SELECT 2 : Is NOT AVAILABLE ?*)						SEL(GVL.IOVD.Z_Semi_Aut_Insu_Tst.na,
(*SELECT 3 : Is ERROR active ?*)						SEL(GVL.IOVD.Z_Semi_Aut_Insu_Tst.e,
(*DEFAULT VALUE assignment*)							0,
(*ERROR is active*)										16#FE),
(*NOT AVAILABLE is active*)								16#FF),
(*Transmission is VALID*)								USINT_TO_BYTE(REAL_TO_USINT((GVL.IOVD.Z_Semi_Aut_Insu_Tst.x))));
{endregion}

{region " SIGNAL AREA : NAME->S_Insu_Tst_Ok LENGTH->1 STARTBIT :24"}
_FB_CanTx_Message_Unpack_485.S_Bit_24		:= GVL.IOVD.S_Insu_Tst_Ok.x AND GVL.IOVD.S_Insu_Tst_Ok.v;
{endregion}

{region " SIGNAL AREA : NAME->S_Man_Insu_Meas_Actv LENGTH->1 STARTBIT :25"}
_FB_CanTx_Message_Unpack_485.S_Bit_25		:= GVL.IOVD.S_Man_Insu_Meas_Actv.x AND GVL.IOVD.S_Man_Insu_Meas_Actv.v;
{endregion}

{region " SIGNAL AREA : NAME->S_Aut_Insu_Meas_Actv LENGTH->1 STARTBIT :26"}
_FB_CanTx_Message_Unpack_485.S_Bit_27		:= GVL.IOVD.S_Aut_Insu_Meas_Actv.x AND GVL.IOVD.S_Aut_Insu_Meas_Actv.v;
{endregion}

_FB_CanTx_Message_Unpack_485.S_Bit_5		:= TRUE;
_FB_CanTx_Message_Unpack_485.S_Bit_6		:= TRUE;
_FB_CanTx_Message_Unpack_485.S_Bit_7		:= TRUE;
_FB_CanTx_Message_Unpack_485.S_Bit_29		:= TRUE;
_FB_CanTx_Message_Unpack_485.S_Bit_30		:= TRUE;
_FB_CanTx_Message_Unpack_485.S_Bit_31		:= TRUE;
_FB_CanTx_Message_Unpack_485.X_Byte_4		:= 16#FF;
_FB_CanTx_Message_Unpack_485.X_Byte_5		:= 16#FF;
_FB_CanTx_Message_Unpack_485.X_Byte_6		:= 16#FF;
_FB_CanTx_Message_Unpack_485.X_Byte_7		:= 16#FF;

_FB_CanTx_Message_Unpack_485 (		C_Enable		:= GVL.IOVD.C_En_Isolation_Status_0X485,
     								Obj_CAN			:= ADR(GVL.IC.Obj_CAN0),
     								X_MsgID			:= 16#485,
     								Tm_CycleTime	:= TIME#250MS,
     								N_Msg_Dlc		:= 8,
     								S_Extended		:= 0,
     								S_Sent_Ok   	=> GVL.IOVD.S_SentOk_Isolation_Status_0X485);
{endregion}
//-----------------------------------------------------------------------------------------------------------------------------
//-----------------------------------------------------------------------------------------------------------------------------
{region " MESSAGE AREA :Arac_Genel_Istatistik- ID:4C2"}

{region " SIGNAL AREA : NAME->X_Spd_TCU LENGTH->8 STARTBIT :0"}
_FB_CanTx_Message_4C2.X_Byte_0							:=
(*SELECT 1 : Is data valid and range is not exceed?*)	SEL((GVL.IOVD.X_Spd_TCU.v AND NOT GVL.IOVD.X_Spd_TCU.RangeExcd),
(*SELECT 2 : Is NOT AVAILABLE ?*)						SEL(GVL.IOVD.X_Spd_TCU.na,
(*SELECT 3 : Is ERROR active ?*)						SEL(GVL.IOVD.X_Spd_TCU.e,
(*DEFAULT VALUE assignment*)							0,
(*ERROR is active*)										16#FE),
(*NOT AVAILABLE is active*)								16#FF),
(*Transmission is VALID*)								USINT_TO_BYTE(REAL_TO_USINT((GVL.IOVD.X_Spd_TCU.x))));
{endregion}

{region " SIGNAL AREA : NAME->X_Spd_EBS LENGTH->8 STARTBIT :8"}
_FB_CanTx_Message_4C2.X_Byte_1							:=
(*SELECT 1 : Is data valid and range is not exceed?*)	SEL((GVL.IOVD.X_Spd_EBS.v AND NOT GVL.IOVD.X_Spd_EBS.RangeExcd),
(*SELECT 2 : Is NOT AVAILABLE ?*)						SEL(GVL.IOVD.X_Spd_EBS.na,
(*SELECT 3 : Is ERROR active ?*)						SEL(GVL.IOVD.X_Spd_EBS.e,
(*DEFAULT VALUE assignment*)							0,
(*ERROR is active*)										16#FE),
(*NOT AVAILABLE is active*)								16#FF),
(*Transmission is VALID*)								USINT_TO_BYTE(REAL_TO_USINT((GVL.IOVD.X_Spd_EBS.x))));
{endregion}

{region " SIGNAL AREA : NAME->X_SOC LENGTH->8 STARTBIT :16"}
_FB_CanTx_Message_4C2.X_Byte_2							:=
(*SELECT 1 : Is data valid and range is not exceed?*)	SEL((GVL.IOVD.X_SOC.v AND NOT GVL.IOVD.X_SOC.RangeExcd),
(*SELECT 2 : Is NOT AVAILABLE ?*)						SEL(GVL.IOVD.X_SOC.na,
(*SELECT 3 : Is ERROR active ?*)						SEL(GVL.IOVD.X_SOC.e,
(*DEFAULT VALUE assignment*)							0,
(*ERROR is active*)										16#FE),
(*NOT AVAILABLE is active*)								16#FF),
(*Transmission is VALID*)								USINT_TO_BYTE(REAL_TO_USINT((GVL.IOVD.X_SOC.x))));
{endregion}

{region " SIGNAL AREA : NAME->X_SOH LENGTH->8 STARTBIT :24"}
_FB_CanTx_Message_4C2.X_Byte_3							:=
(*SELECT 1 : Is data valid and range is not exceed?*)	SEL((GVL.IOVD.X_SOH.v AND NOT GVL.IOVD.X_SOH.RangeExcd),
(*SELECT 2 : Is NOT AVAILABLE ?*)						SEL(GVL.IOVD.X_SOH.na,
(*SELECT 3 : Is ERROR active ?*)						SEL(GVL.IOVD.X_SOH.e,
(*DEFAULT VALUE assignment*)							0,
(*ERROR is active*)										16#FE),
(*NOT AVAILABLE is active*)								16#FF),
(*Transmission is VALID*)								USINT_TO_BYTE(REAL_TO_USINT((GVL.IOVD.X_SOH.x))));
{endregion}

{region " SIGNAL AREA : NAME->X_Accl LENGTH->16 STARTBIT :32"}
_FB_UNPACK_WORD_TO_BYTE_24 (	X_WORD_0	:= 
(*SELECT 1 : Is data valid and range is not exceed?*)	SEL((GVL.IOVD.X_Accl.v AND NOT GVL.IOVD.X_Accl.RangeExcd),
(*SELECT 2 : Is NOT AVAILABLE ?*)						SEL(GVL.IOVD.X_Accl.na,
(*SELECT 3 : Is ERROR active ?*)						SEL(GVL.IOVD.X_Accl.e,
(*DEFAULT VALUE assignment*)							UINT_TO_WORD(REAL_TO_UINT((32)/0.001)),
(*ERROR is active*)										16#FEFE),
(*NOT AVAILABLE is active*)								16#FFFF),
(*Transmission is VALID*)								UINT_TO_WORD(REAL_TO_UINT((GVL.IOVD.X_Accl.x + 32)/0.001))),
								X_BYTE_0	=> _FB_CanTx_Message_4C2.X_Byte_4,
								X_BYTE_1	=> _FB_CanTx_Message_4C2.X_Byte_5);
{endregion}

{region " SIGNAL AREA : NAME->X_Cosu_Avg LENGTH->16 STARTBIT :48"}
_FB_UNPACK_WORD_TO_BYTE_25 (
		X_WORD_0										:= 
(*SELECT 1 : Is data valid and range is not exceed?*)	SEL((GVL.IOVD.X_Cosu_Avg.v AND NOT GVL.IOVD.X_Cosu_Avg.RangeExcd),
(*SELECT 2 : Is NOT AVAILABLE ?*)						SEL(GVL.IOVD.X_Cosu_Avg.na,
(*SELECT 3 : Is ERROR active ?*)						SEL(GVL.IOVD.X_Cosu_Avg.e,
(*DEFAULT VALUE assignment*)							0,
(*ERROR is active*)										16#FEFE),
(*NOT AVAILABLE is active*)								16#FFFF),
(*Transmission is VALID*)								UINT_TO_WORD(REAL_TO_UINT((GVL.IOVD.X_Cosu_Avg.x)/0.001))),
		X_BYTE_0										=> _FB_CanTx_Message_4C2.X_Byte_6,
		X_BYTE_1										=> _FB_CanTx_Message_4C2.X_Byte_7);
{endregion}

_FB_CanTx_Message_4C2 (		C_Enable		:= GVL.IOVD.C_En_Arac_Genel_Istatistik_0X4C2,
     						Obj_CAN			:= ADR(GVL.IC.Obj_CAN0),
     						X_MsgID			:= 16#4C2,
     						Tm_CycleTime	:= TIME#250MS,
     						N_Msg_Dlc		:= 8,
     						S_Extended		:= 0,
     						S_Sent_Ok   	=> GVL.IOVD.S_SentOk_Arac_Genel_Istatistik_0X4C2);
{endregion}
//-----------------------------------------------------------------------------------------------------------------------------
//-----------------------------------------------------------------------------------------------------------------------------
{region " MESSAGE AREA :Temel_Durum- ID:99"}

{region " SIGNAL AREA : NAME->N_ECU_Lf LENGTH->8 STARTBIT :0"}
_FB_CanTx_Message_Unpack_99.X_Byte_0		:=
(*SELECT 1 : Is data valid and range is not exceed?*)	SEL((GVL.IOVD.N_ECU_Lf.v AND NOT GVL.IOVD.N_ECU_Lf.RangeExcd),
(*SELECT 2 : Is NOT AVAILABLE ?*)						SEL(GVL.IOVD.N_ECU_Lf.na,
(*SELECT 3 : Is ERROR active ?*)						SEL(GVL.IOVD.N_ECU_Lf.e,
(*DEFAULT VALUE assignment*)							0,
(*ERROR is active*)										16#FE),
(*NOT AVAILABLE is active*)								16#FF),
(*Transmission is VALID*)								USINT_TO_BYTE(GVL.IOVD.N_ECU_Lf.x ));

{endregion}

// PR1006_SRS_001391_TIMTRO
{region " SIGNAL AREA : NAME->S_Sw_Up_Avl LENGTH->2 STARTBIT :8"}
_FB_CanTx_Message_Unpack_99.S_Bit_8		:=	 (GVL.IOVD.S_Sw_Up_Avl.x OR GVL.IOVD.S_Sw_Up_Avl.na) AND NOT GVL.IOVD.S_Sw_Up_Avl.e; 
_FB_CanTx_Message_Unpack_99.S_Bit_9		:=	 NOT GVL.IOVD.S_Sw_Up_Avl.v OR GVL.IOVD.S_Sw_Up_Avl.na OR GVL.IOVD.S_Sw_Up_Avl.e; 

{endregion}

{region " SIGNAL AREA : NAME->S_EH_Rd_Avl LENGTH->2 STARTBIT :10"}
_FB_CanTx_Message_Unpack_99.S_Bit_10		:=	 (GVL.IOVD.S_EH_Rd_Avl.x OR GVL.IOVD.S_EH_Rd_Avl.na) AND NOT GVL.IOVD.S_EH_Rd_Avl.e; 
_FB_CanTx_Message_Unpack_99.S_Bit_11		:=	 NOT GVL.IOVD.S_EH_Rd_Avl.v OR GVL.IOVD.S_EH_Rd_Avl.na OR GVL.IOVD.S_EH_Rd_Avl.e; 

{endregion}

{region " SIGNAL AREA : NAME->S_Tst_Avl LENGTH->2 STARTBIT :12"}
_FB_CanTx_Message_Unpack_99.S_Bit_12		:=	 (GVL.IOVD.S_Tst_Avl.x OR GVL.IOVD.S_Tst_Avl.na) AND NOT GVL.IOVD.S_Tst_Avl.e; 
_FB_CanTx_Message_Unpack_99.S_Bit_13		:=	 NOT GVL.IOVD.S_Tst_Avl.v OR GVL.IOVD.S_Tst_Avl.na OR GVL.IOVD.S_Tst_Avl.e; 

{endregion}

{region " SIGNAL AREA : NAME->S_Para_Up_Avl LENGTH->2 STARTBIT :14"}
_FB_CanTx_Message_Unpack_99.S_Bit_14		:=	 (GVL.IOVD.S_Para_Up_Avl.x OR GVL.IOVD.S_Para_Up_Avl.na) AND NOT GVL.IOVD.S_Para_Up_Avl.e; 
_FB_CanTx_Message_Unpack_99.S_Bit_15		:=	 NOT GVL.IOVD.S_Para_Up_Avl.v OR GVL.IOVD.S_Para_Up_Avl.na OR GVL.IOVD.S_Para_Up_Avl.e; 

{endregion}

{region " SIGNAL AREA : NAME->C_ECU_Rst LENGTH->2 STARTBIT :16"}
_FB_CanTx_Message_Unpack_99.S_Bit_16		:=	 (GVL.IOVD.C_ECU_Rst.x OR GVL.IOVD.C_ECU_Rst.na) AND NOT GVL.IOVD.C_ECU_Rst.e; 
_FB_CanTx_Message_Unpack_99.S_Bit_17		:=	 NOT GVL.IOVD.C_ECU_Rst.v OR GVL.IOVD.C_ECU_Rst.na OR GVL.IOVD.C_ECU_Rst.e; 

{endregion}
{region " SIGNAL AREA : NAME->S_Brk_Tst_Mode LENGTH->2 STARTBIT :18"}
_FB_CanTx_Message_Unpack_99.S_Bit_18		:=	 (GVL.IOVD.S_Brk_Tst_Mode.x OR GVL.IOVD.S_Brk_Tst_Mode.na) AND NOT GVL.IOVD.S_Brk_Tst_Mode.e; 
_FB_CanTx_Message_Unpack_99.S_Bit_19		:=	 NOT GVL.IOVD.S_Brk_Tst_Mode.v OR GVL.IOVD.S_Brk_Tst_Mode.na OR GVL.IOVD.S_Brk_Tst_Mode.e; 

{endregion}
		  
{region " SIGNAL AREA : NAME->Z_Vh_Typ LENGTH->8 STARTBIT :32"}
_FB_CanTx_Message_Unpack_99.X_Byte_4		:=
(*SELECT 1 : Is data valid and range is not exceed?*)	SEL((GVL.IOVD.Z_Vh_Typ.v AND NOT GVL.IOVD.Z_Vh_Typ.RangeExcd),
(*SELECT 2 : Is NOT AVAILABLE ?*)						SEL(GVL.IOVD.Z_Vh_Typ.na,
(*SELECT 3 : Is ERROR active ?*)						SEL(GVL.IOVD.Z_Vh_Typ.e,
(*DEFAULT VALUE assignment*)							0,
(*ERROR is active*)										16#E),
(*NOT AVAILABLE is active*)								16#F),
(*Transmission is VALID*)								GVL.IOVD.Z_Vh_Typ.x);
{endregion}

// PR1006_SRS_001386_TIMTRO
{region " SIGNAL AREA : NAME->X_Prj_No LENGTH->16 STARTBIT->48}
_FB_UNPACK_WORD_TO_BYTE_30	(	X_Word_0				:=  
(*SELECT 1: Is data valid and range is not exceed?*)	SEL((GVL.IOVD.X_Prj_No.v AND NOT GVL.IOVD.X_Prj_No.RangeExcd),
(*SELECT 2: Is NOT AVAILABLE ?*)						SEL(GVL.IOVD.X_Prj_No.na,
(*SELECT 3: Is ERROR active ?*)							SEL(GVL.IOVD.X_Prj_No.e,
(*DEFAULT VALUE assignment*)							1000,
(*ERROR is active*)										16#FEFF),
(*NOT AVAILABLE is active*)								16#FFFF),
(*Transmission is VALID*)								UINT_TO_WORD(REAL_TO_UINT(GVL.IOVD.X_Prj_No.x))),
														X_Byte_0=> _FB_CanTx_Message_Unpack_99.X_Byte_6,
														X_Byte_1=> _FB_CanTx_Message_Unpack_99.X_Byte_7);
{endregion}
  
_FB_CanTx_Message_Unpack_99.S_Bit_22:=TRUE;
_FB_CanTx_Message_Unpack_99.S_Bit_23:=TRUE;
_FB_CanTx_Message_Unpack_99.X_Byte_3:=16#FF;
_FB_CanTx_Message_Unpack_99.X_Byte_5:=16#FF;
_FB_CanTx_Message_Unpack_99(
     C_Enable:= GVL.IOVD.C_En_Temel_Durum_0X99,
     Obj_CAN:= ADR(GVL.IC.Obj_CAN0),
     X_MsgID:= 16#99,
     Tm_CycleTime:= TIME#250ms,
     N_Msg_Dlc:=8,
     S_Extended:= 0,
     S_Sent_Ok   => GVL.IOVD.S_SentOk_Temel_Durum_0X99);
{endregion}
	 
	 
{region " MESSAGE AREA :Olay_Durum- ID:500"}

// PR1006_SRS_001881_TIMTRO
{region " SIGNAL AREA : NAME->X_Tot_TypA_Evnt LENGTH->16 STARTBIT :0"}
_FB_UNPACK_WORD_TO_BYTE_28(
		X_WORD_0:= 
(*SELECT 1 : Is data valid and range is not exceed?*)	SEL((GVL.IOVD.X_Tot_TypA_Evnt.v AND NOT GVL.IOVD.X_Tot_TypA_Evnt.RangeExcd),
(*SELECT 2 : Is NOT AVAILABLE ?*)						SEL(GVL.IOVD.X_Tot_TypA_Evnt.na,
(*SELECT 3 : Is ERROR active ?*)						SEL(GVL.IOVD.X_Tot_TypA_Evnt.e,
(*DEFAULT VALUE assignment*)							 0,
(*ERROR is active*)										16#FEFE),
(*NOT AVAILABLE is active*)								16#FFFF),
(*Transmission is VALID*)								UINT_TO_WORD(REAL_TO_UINT((GVL.IOVD.X_Tot_TypA_Evnt.x)))),
		X_BYTE_0=> _FB_CanTx_Message_500.X_Byte_0,
		X_BYTE_1=> _FB_CanTx_Message_500.X_Byte_1);
{endregion}

// PR1006_SRS_001881_TIMTRO
{region " SIGNAL AREA : NAME->X_Tot_TypB_Evnt LENGTH->16 STARTBIT :16"}
_FB_UNPACK_WORD_TO_BYTE_29(
		X_WORD_0:= 
(*SELECT 1 : Is data valid and range is not exceed?*)	SEL((GVL.IOVD.X_Tot_TypB_Evnt.v AND NOT GVL.IOVD.X_Tot_TypB_Evnt.RangeExcd),
(*SELECT 2 : Is NOT AVAILABLE ?*)						SEL(GVL.IOVD.X_Tot_TypB_Evnt.na,
(*SELECT 3 : Is ERROR active ?*)						SEL(GVL.IOVD.X_Tot_TypB_Evnt.e,
(*DEFAULT VALUE assignment*)							 0,
(*ERROR is active*)										16#FEFE),
(*NOT AVAILABLE is active*)								16#FFFF),
(*Transmission is VALID*)								UINT_TO_WORD(REAL_TO_UINT((GVL.IOVD.X_Tot_TypB_Evnt.x)))),
		X_BYTE_0=> _FB_CanTx_Message_500.X_Byte_2,
		X_BYTE_1=> _FB_CanTx_Message_500.X_Byte_3);
{endregion}
		  
_FB_CanTx_Message_500.X_Byte_4 := 16#FF;
_FB_CanTx_Message_500.X_Byte_5 := 16#FF;
_FB_CanTx_Message_500.X_Byte_6 := 16#FF;
_FB_CanTx_Message_500.X_Byte_7 := 16#FF;

_FB_CanTx_Message_500(	C_Enable := GVL.IOVD.C_En_Olay_Durum_0X500,
		 				Obj_CAN := ADR(GVL.IC.Obj_CAN0),
						X_MsgID := 16#500,
						Tm_CycleTime := T#250MS,
						N_Msg_Dlc := 8,
						S_Extended := FALSE,
						S_Sent_Ok => GVL.IOVD.S_SentOk_Olay_Durum_0X500);

{endregion}
//-----------------------------------------------------------------------------------------------------------------------------
          
END_PROGRAM
